C01816=1094.495,429.613,397.808,178.819,24.459,153.656
C01817=1094.490,429.367,397.851,178.817,24.448,153.653
C01818=1094.483,429.120,397.893,178.813,24.437,153.651
C01819=1094.477,428.875,397.935,178.811,24.426,153.649
C01820=1094.470,428.628,397.977,178.808,24.416,153.646
C01821=1094.464,428.382,398.019,178.805,24.405,153.644
C01822=1094.457,428.135,398.061,178.802,24.394,153.642
C01823=1094.451,427.889,398.102,178.799,24.383,153.639
C01824=1094.445,427.643,398.145,178.797,24.373,153.637
C01825=1094.439,427.397,398.186,178.793,24.362,153.635
C01826=1094.433,427.150,398.228,178.791,24.352,153.633
C01827=1094.426,426.904,398.270,178.788,24.342,153.630
C01828=1094.420,426.658,398.312,178.785,24.331,153.628
C01829=1094.413,426.411,398.354,178.782,24.320,153.626
C01830=1094.407,426.165,398.395,178.779,24.310,153.624
C01831=1094.401,425.919,398.437,178.776,24.300,153.622
C01832=1094.395,425.672,398.478,178.774,24.289,153.619
C01833=1094.389,425.443,398.517,178.771,24.280,153.617
C01834=1094.384,425.215,398.556,178.768,24.270,153.615
C01835=1094.378,424.987,398.594,178.766,24.261,153.613
C01836=1094.372,424.758,398.633,178.763,24.251,153.611
C01837=1094.366,424.529,398.671,178.760,24.242,153.609
C01838=1094.360,424.301,398.710,178.757,24.232,153.607
C01839=1094.355,424.073,398.748,178.755,24.223,153.605
C01840=1094.349,423.844,398.787,178.752,24.214,153.603
C01841=1094.344,423.598,398.828,178.749,24.204,153.601
C01842=1094.337,423.351,398.870,178.746,24.194,153.599
C01843=1094.330,423.105,398.911,178.744,24.184,153.597
C01844=1094.324,422.859,398.953,178.741,24.174,153.595
C01845=1094.319,422.612,398.993,178.738,24.164,153.593
C01846=1094.312,422.365,399.035,178.734,24.154,153.591
C01847=1094.306,422.119,399.077,178.732,24.144,153.589
C01848=1094.300,421.873,399.117,178.729,24.134,153.587
C01849=1094.294,421.627,399.158,178.726,24.125,153.585
C01850=1094.287,421.380,399.200,178.723,24.115,153.583
C01851=1094.281,421.134,399.241,178.720,24.105,153.581
C01852=1094.275,420.887,399.282,178.717,24.095,153.579
C01853=1094.269,420.641,399.323,178.714,24.086,153.577
C01854=1094.263,420.393,399.364,178.712,24.076,153.575
C01855=1094.256,420.147,399.405,178.709,24.067,153.573
C01856=1094.250,419.901,399.447,178.706,24.057,153.571
C01857=1094.245,419.654,399.487,178.703,24.048,153.569
C01858=1094.238,419.408,399.528,178.700,24.038,153.567
C01859=1094.232,419.161,399.569,178.697,24.029,153.565
C01860=1094.225,418.914,399.609,178.694,24.019,153.563
C01861=1094.219,418.668,399.651,178.691,24.010,153.561
C01862=1094.214,418.421,399.692,178.689,24.000,153.559
C01863=1094.207,418.175,399.732,178.686,23.991,153.557
C01864=1094.201,417.929,399.773,178.683,23.982,153.555
C01865=1094.195,417.682,399.813,178.680,23.972,153.553
C01866=1094.189,417.436,399.855,178.677,23.963,153.551
C01867=1094.183,417.188,399.896,178.675,23.954,153.549
C01868=1094.176,416.942,399.936,178.672,23.945,153.548
C01869=1094.171,416.695,399.977,178.669,23.936,153.546
C01870=1094.164,416.449,400.018,178.666,23.926,153.544
C01871=1094.158,416.202,400.058,178.663,23.918,153.542
C01872=1094.152,415.956,400.099,178.660,23.908,153.540
C01873=1094.146,415.709,400.139,178.657,23.899,153.538
C01874=1094.140,415.462,400.179,178.654,23.890,153.536
C01875=1094.134,415.216,400.220,178.652,23.882,153.535
C01876=1094.128,414.969,400.260,178.649,23.873,153.533
C01877=1094.122,414.723,400.300,178.646,23.864,153.531
C01878=1094.114,414.476,400.342,178.643,23.855,153.529
C01879=1094.109,414.229,400.382,178.640,23.846,153.527
C01880=1094.102,413.983,400.423,178.636,23.837,153.526
C01881=1094.096,413.735,400.462,178.634,23.828,153.524
C01882=1094.091,413.489,400.503,178.631,23.820,153.522
C01883=1094.084,413.242,400.543,178.628,23.811,153.520
C01884=1094.078,412.996,400.583,178.625,23.802,153.519
C01885=1094.071,412.749,400.623,178.623,23.794,153.517
C01886=1094.066,412.502,400.664,178.620,23.785,153.515
C01887=1094.059,412.256,400.704,178.617,23.776,153.513
C01888=1094.053,412.009,400.744,178.614,23.768,153.512
C01889=1094.048,411.788,400.779,178.611,23.760,153.510
C01890=1094.043,411.567,400.816,178.609,23.753,153.509
C01891=1094.038,411.345,400.852,178.606,23.745,153.507
C01892=1094.032,411.125,400.888,178.604,23.737,153.506
C01893=1094.026,410.904,400.924,178.601,23.730,153.504
C01894=1094.021,410.682,400.959,178.599,23.722,153.503
C01895=1094.015,410.461,400.996,178.595,23.714,153.501
C01896=1094.011,410.240,401.031,178.593,23.706,153.499
C01897=1094.004,409.993,401.071,178.591,23.698,153.498
C01898=1093.998,409.746,401.111,178.588,23.690,153.496
C01899=1093.992,409.500,401.151,178.584,23.681,153.495
C01900=1093.986,409.253,401.192,178.582,23.673,153.493
C01901=1093.980,409.006,401.231,178.579,23.665,153.491
C01902=1093.974,408.759,401.271,178.576,23.656,153.490
C01903=1093.968,408.513,401.310,178.574,23.648,153.488
C01904=1093.962,408.266,401.350,178.570,23.640,153.486
C01905=1093.956,408.019,401.390,178.568,23.632,153.485
C01906=1093.949,407.773,401.430,178.565,23.624,153.483
C01907=1093.943,407.525,401.469,178.561,23.616,153.482
C01908=1093.938,407.279,401.509,178.559,23.607,153.480
C01909=1093.932,407.032,401.549,178.556,23.599,153.478
C01910=1093.926,406.785,401.589,178.554,23.591,153.477
C01911=1093.920,406.538,401.628,178.550,23.583,153.475
C01912=1093.914,406.291,401.668,178.547,23.575,153.474
C01913=1093.908,406.045,401.707,178.545,23.567,153.472
C01914=1093.902,405.798,401.747,178.542,23.559,153.470
C01915=1093.895,405.551,401.786,178.539,23.551,153.469
C01916=1093.889,405.304,401.826,178.536,23.543,153.467
C01917=1093.883,405.058,401.865,178.533,23.536,153.466
C01918=1093.877,404.811,401.904,178.530,23.528,153.464
C01919=1093.871,404.564,401.944,178.528,23.520,153.463
C01920=1093.865,404.317,401.983,178.524,23.512,153.461
C01921=1093.859,404.071,402.023,178.522,23.504,153.460
C01922=1093.853,403.824,402.062,178.519,23.497,153.458
C01923=1093.847,403.577,402.101,178.516,23.489,153.457
C01924=1093.841,403.330,402.140,178.513,23.481,153.455
C01925=1093.835,403.083,402.180,178.510,23.474,153.454
C01926=1093.829,402.836,402.219,178.507,23.466,153.452
C01927=1093.823,402.590,402.258,178.505,23.458,153.451
C01928=1093.817,402.343,402.297,178.501,23.450,153.449
C01929=1093.811,402.096,402.336,178.499,23.443,153.448
C01930=1093.805,401.849,402.375,178.496,23.435,153.446
C01931=1093.799,401.602,402.415,178.493,23.428,153.445
C01932=1093.792,401.355,402.454,178.490,23.421,153.444
C01933=1093.787,401.108,402.492,178.487,23.412,153.442
C01934=1093.781,400.861,402.532,178.485,23.405,153.441
C01935=1093.775,400.614,402.571,178.482,23.398,153.439
C01936=1093.769,400.368,402.609,178.479,23.390,153.438
C01937=1093.763,400.121,402.649,178.476,23.383,153.437
C01938=1093.757,399.874,402.688,178.473,23.376,153.435
C01939=1093.751,399.627,402.726,178.470,23.368,153.434
C01940=1093.745,399.380,402.765,178.468,23.361,153.432
C01941=1093.739,399.133,402.805,178.464,23.353,153.431
C01942=1093.733,398.886,402.843,178.462,23.346,153.430
C01943=1093.727,398.639,402.882,178.459,23.339,153.428
C01944=1093.720,398.393,402.921,178.456,23.332,153.427
C01945=1093.715,398.172,402.956,178.453,23.325,153.426
C01946=1093.710,397.951,402.990,178.451,23.319,153.424
C01947=1093.704,397.730,403.024,178.448,23.312,153.423
C01948=1093.700,397.509,403.059,178.446,23.306,153.422
C01949=1093.694,397.289,403.093,178.443,23.299,153.421
C01950=1093.688,397.068,403.128,178.441,23.293,153.420
C01951=1093.683,396.847,403.163,178.438,23.287,153.418
C01952=1093.678,396.626,403.197,178.435,23.280,153.417
C01953=1093.671,396.379,403.236,178.433,23.274,153.416
C01954=1093.666,396.132,403.274,178.430,23.266,153.415
C01955=1093.659,395.885,403.313,178.427,23.259,153.413
C01956=1093.654,395.638,403.351,178.424,23.252,153.412
C01957=1093.647,395.391,403.390,178.421,23.245,153.411
C01958=1093.642,395.144,403.428,178.418,23.238,153.409
C01959=1093.636,394.898,403.467,178.415,23.231,153.408
C01960=1093.630,394.650,403.506,178.413,23.224,153.407
C01961=1093.624,394.404,403.543,178.410,23.217,153.406
C01962=1093.618,394.157,403.582,178.406,23.210,153.404
C01963=1093.612,393.910,403.621,178.404,23.203,153.403
C01964=1093.606,393.663,403.658,178.401,23.197,153.402
C01965=1093.600,393.416,403.697,178.398,23.190,153.401
C01966=1093.594,393.169,403.735,178.395,23.183,153.399
C01967=1093.588,392.922,403.774,178.392,23.176,153.398
C01968=1093.582,392.675,403.811,178.389,23.169,153.397
C01969=1093.576,392.428,403.849,178.387,23.163,153.396
C01970=1093.570,392.181,403.889,178.384,23.156,153.394
C01971=1093.564,391.934,403.926,178.380,23.149,153.393
C01972=1093.558,391.688,403.964,178.378,23.142,153.392
C01973=1093.552,391.440,404.002,178.375,23.136,153.391
C01974=1093.546,391.193,404.040,178.372,23.130,153.390
C01975=1093.540,390.947,404.078,178.369,23.123,153.388
C01976=1093.534,390.699,404.116,178.366,23.116,153.387
C01977=1093.528,390.452,404.154,178.363,23.110,153.386
C01978=1093.522,390.206,404.193,178.360,23.103,153.385
C01979=1093.516,389.959,404.231,178.357,23.096,153.384
C01980=1093.510,389.712,404.268,178.355,23.090,153.383
C01981=1093.504,389.465,404.306,178.351,23.083,153.381
C01982=1093.498,389.218,404.344,178.348,23.076,153.380
C01983=1093.491,388.971,404.382,178.345,23.070,153.379
C01984=1093.486,388.724,404.419,178.343,23.064,153.378
C01985=1093.480,388.477,404.457,178.340,23.057,153.377
C01986=1093.474,388.230,404.495,178.337,23.051,153.376
C01987=1093.468,387.983,404.532,178.333,23.044,153.375
C01988=1093.462,387.736,404.571,178.331,23.038,153.373
C01989=1093.456,387.489,404.608,178.328,23.031,153.372
C01990=1093.450,387.242,404.646,178.325,23.025,153.371
C01991=1093.444,386.995,404.683,178.322,23.019,153.370
C01992=1093.438,386.748,404.721,178.319,23.013,153.369
C01993=1093.432,386.502,404.759,178.316,23.006,153.368
C01994=1093.426,386.254,404.797,178.314,23.000,153.367
C01995=1093.420,386.007,404.834,178.310,22.993,153.366
C01996=1093.414,385.760,404.872,178.307,22.987,153.365
C01997=1093.408,385.513,404.909,178.304,22.981,153.363
C01998=1093.402,385.267,404.947,178.301,22.975,153.362
C01999=1093.397,385.019,404.984,178.298,22.969,153.361
C02000=1093.391,384.772,405.022,178.296,22.962,153.360
C02001=1093.386,384.558,405.054,178.294,22.957,153.359
C02002=1093.381,384.343,405.087,178.290,22.951,153.358
C02003=1093.376,384.129,405.120,178.288,22.946,153.357
C02004=1093.371,383.915,405.152,178.285,22.940,153.356
C02005=1093.365,383.700,405.184,178.283,22.935,153.356
C02006=1093.361,383.486,405.217,178.281,22.930,153.355
C02007=1093.355,383.272,405.249,178.278,22.924,153.354
C02008=1093.351,383.057,405.281,178.276,22.919,153.353
C02009=1093.345,382.811,405.319,178.273,22.913,153.352
C02010=1093.339,382.563,405.356,178.270,22.907,153.351
C02011=1093.332,382.316,405.393,178.267,22.901,153.350
C02012=1093.326,382.069,405.431,178.264,22.895,153.349
C02013=1093.321,381.821,405.468,178.261,22.889,153.348
C02014=1093.314,381.575,405.505,178.258,22.883,153.347
C02015=1093.308,381.328,405.542,178.255,22.877,153.346
C02016=1093.303,381.080,405.579,178.252,22.871,153.345
C02017=1093.296,380.834,405.616,178.249,22.866,153.344
C02018=1093.291,380.587,405.653,178.245,22.859,153.343
C02019=1093.285,380.339,405.690,178.242,22.853,153.342
C02020=1093.278,380.093,405.727,178.239,22.847,153.341
C02021=1093.273,379.845,405.764,178.237,22.841,153.340
C02022=1093.267,379.598,405.801,178.234,22.836,153.339
C02023=1093.261,379.351,405.838,178.231,22.830,153.338
C02024=1093.255,379.104,405.875,178.228,22.824,153.337
C02025=1093.249,378.857,405.913,178.226,22.818,153.336
C02026=1093.243,378.610,405.949,178.222,22.813,153.335
C02027=1093.237,378.362,405.986,178.219,22.807,153.334
C02028=1093.231,378.115,406.023,178.217,22.801,153.333
C02029=1093.225,377.868,406.060,178.213,22.796,153.332
C02030=1093.220,377.621,406.097,178.210,22.790,153.331
C02031=1093.213,377.374,406.133,178.208,22.784,153.330
C02032=1093.208,377.127,406.170,178.204,22.778,153.329
C02033=1093.202,376.880,406.206,178.202,22.772,153.328
C02034=1093.197,376.633,406.243,178.198,22.767,153.327
C02035=1093.191,376.385,406.280,178.196,22.761,153.326
C02036=1093.185,376.138,406.317,178.192,22.755,153.325
C02037=1093.179,375.891,406.354,178.189,22.749,153.324
C02038=1093.173,375.644,406.390,178.186,22.744,153.323
C02039=1093.167,375.396,406.427,178.183,22.738,153.323
C02040=1093.161,375.150,406.463,178.180,22.732,153.322
C02041=1093.156,374.903,406.500,178.177,22.727,153.321
C02042=1093.149,374.656,406.537,178.175,22.722,153.320
C02043=1093.144,374.408,406.574,178.172,22.716,153.319
C02044=1093.138,374.160,406.610,178.169,22.710,153.318
C02045=1093.132,373.913,406.647,178.166,22.705,153.317
C02046=1093.126,373.666,406.683,178.163,22.699,153.316
C02047=1093.120,373.420,406.719,178.160,22.694,153.315
C02048=1093.115,373.172,406.756,178.157,22.688,153.315
C02049=1093.108,372.925,406.792,178.154,22.683,153.314
C02050=1093.102,372.678,406.828,178.150,22.677,153.313
C02051=1093.096,372.431,406.865,178.147,22.672,153.312
C02052=1093.091,372.183,406.901,178.145,22.667,153.311
C02053=1093.084,371.936,406.938,178.142,22.661,153.310
C02054=1093.078,371.689,406.974,178.139,22.656,153.309
C02055=1093.073,371.441,407.010,178.136,22.650,153.309
C02056=1093.067,371.194,407.047,178.133,22.645,153.308
C02057=1093.057,370.793,407.105,178.128,22.636,153.306
C02058=1093.048,370.391,407.164,178.123,22.627,153.305
C02059=1093.038,369.990,407.223,178.119,22.619,153.304
C02060=1093.029,369.590,407.281,178.114,22.610,153.302
C02061=1093.023,369.342,407.317,178.111,22.605,153.301
C02062=1093.017,369.094,407.353,178.107,22.600,153.301
C02063=1093.011,368.847,407.390,178.104,22.594,153.300
C02064=1093.005,368.600,407.425,178.101,22.589,153.299
C02065=1092.999,368.353,407.462,178.099,22.584,153.298
C02066=1092.993,368.105,407.497,178.096,22.579,153.297
C02067=1092.988,367.858,407.533,178.092,22.574,153.297
C02068=1092.982,367.611,407.570,178.089,22.568,153.296
C02069=1092.976,367.363,407.606,178.086,22.563,153.295
C02070=1092.971,367.116,407.641,178.084,22.558,153.294
C02071=1092.964,366.869,407.677,178.081,22.553,153.293
C02072=1092.958,366.622,407.713,178.077,22.548,153.293
C02073=1092.954,366.374,407.749,178.074,22.542,153.292
C02074=1092.948,366.127,407.785,178.071,22.537,153.291
C02075=1092.941,365.880,407.821,178.069,22.532,153.290
C02076=1092.936,365.633,407.857,178.066,22.527,153.289
C02077=1092.930,365.385,407.892,178.062,22.522,153.289
C02078=1092.924,365.137,407.928,178.059,22.517,153.288
C02079=1092.918,364.890,407.963,178.056,22.512,153.287
C02080=1092.912,364.643,408.000,178.054,22.507,153.287
C02081=1092.906,364.396,408.036,178.050,22.502,153.286
C02082=1092.900,364.149,408.071,178.047,22.497,153.285
C02083=1092.894,363.901,408.107,178.044,22.491,153.284
C02084=1092.889,363.654,408.142,178.042,22.487,153.284
C02085=1092.883,363.406,408.178,178.038,22.482,153.283
C02086=1092.876,363.159,408.213,178.035,22.477,153.282
C02087=1092.871,362.912,408.248,178.032,22.471,153.281
C02088=1092.865,362.664,408.284,178.029,22.467,153.281
C02089=1092.859,362.417,408.319,178.026,22.462,153.280
C02090=1092.853,362.170,408.355,178.023,22.457,153.279
C02091=1092.847,361.922,408.391,178.020,22.452,153.279
C02092=1092.842,361.675,408.426,178.017,22.447,153.278
C02093=1092.836,361.427,408.462,178.014,22.442,153.277
C02094=1092.831,361.180,408.497,178.011,22.437,153.276
C02095=1092.824,360.932,408.532,178.008,22.433,153.276
C02096=1092.818,360.685,408.567,178.005,22.428,153.275
C02097=1092.812,360.438,408.603,178.002,22.423,153.274
C02098=1092.807,360.191,408.638,177.999,22.418,153.274
C02099=1092.801,359.943,408.674,177.996,22.414,153.273
C02100=1092.795,359.695,408.708,177.993,22.408,153.272
C02101=1092.789,359.448,408.744,177.990,22.403,153.271
C02102=1092.783,359.200,408.779,177.987,22.399,153.271
C02103=1092.778,358.953,408.815,177.984,22.394,153.270
C02104=1092.771,358.705,408.849,177.980,22.389,153.270
C02105=1092.766,358.458,408.885,177.978,22.385,153.269
C02106=1092.760,358.211,408.920,177.975,22.380,153.268
C02107=1092.754,357.963,408.954,177.971,22.375,153.267
C02108=1092.748,357.716,408.990,177.969,22.371,153.267
C02109=1092.739,357.330,409.045,177.963,22.363,153.266
C02110=1092.730,356.944,409.099,177.959,22.356,153.265
C02111=1092.721,356.558,409.154,177.955,22.349,153.264
C02112=1092.712,356.172,409.209,177.950,22.342,153.263
C02113=1092.706,355.925,409.243,177.947,22.337,153.262
C02114=1092.700,355.678,409.278,177.943,22.332,153.261
C02115=1092.695,355.429,409.313,177.941,22.328,153.261
C02116=1092.688,355.183,409.348,177.937,22.323,153.260
C02117=1092.683,354.935,409.383,177.934,22.318,153.260
C02118=1092.677,354.688,409.418,177.932,22.314,153.259
C02119=1092.671,354.440,409.453,177.928,22.309,153.258
C02120=1092.666,354.192,409.488,177.925,22.304,153.258
C02121=1092.659,353.945,409.522,177.922,22.300,153.257
C02122=1092.654,353.697,409.557,177.919,22.295,153.256
C02123=1092.648,353.449,409.592,177.916,22.291,153.256
C02124=1092.642,353.203,409.627,177.913,22.286,153.255
C02125=1092.637,352.955,409.661,177.910,22.282,153.255
C02126=1092.631,352.707,409.696,177.907,22.277,153.254
C02127=1092.625,352.460,409.731,177.904,22.273,153.253
C02128=1092.619,352.212,409.766,177.901,22.269,153.253
C02129=1092.613,351.965,409.800,177.898,22.264,153.252
C02130=1092.608,351.717,409.834,177.894,22.259,153.252
C02131=1092.601,351.470,409.870,177.892,22.255,153.251
C02132=1092.595,351.222,409.904,177.889,22.250,153.250
C02133=1092.586,350.816,409.960,177.884,22.243,153.249
C02134=1092.576,350.409,410.017,177.879,22.236,153.249
C02135=1092.566,350.002,410.074,177.874,22.229,153.248
C02136=1092.557,349.596,410.130,177.869,22.221,153.247
C02137=1092.552,349.348,410.165,177.865,22.217,153.246
C02138=1092.546,349.101,410.199,177.863,22.213,153.245
C02139=1092.540,348.853,410.233,177.859,22.208,153.245
C02140=1092.534,348.605,410.268,177.856,22.204,153.244
C02141=1092.529,348.358,410.302,177.853,22.199,153.244
C02142=1092.523,348.111,410.336,177.851,22.195,153.243
C02143=1092.518,347.863,410.371,177.847,22.191,153.243
C02144=1092.511,347.615,410.405,177.844,22.187,153.242
C02145=1092.505,347.368,410.439,177.841,22.182,153.242
C02146=1092.500,347.120,410.474,177.838,22.178,153.241
C02147=1092.494,346.873,410.508,177.835,22.174,153.241
C02148=1092.488,346.625,410.542,177.832,22.169,153.240
C02149=1092.482,346.377,410.576,177.829,22.165,153.239
C02150=1092.477,346.129,410.610,177.825,22.161,153.239
C02151=1092.471,345.882,410.644,177.823,22.157,153.238
C02152=1092.465,345.635,410.678,177.819,22.152,153.238
C02153=1092.459,345.387,410.713,177.817,22.148,153.237
C02154=1092.453,345.139,410.746,177.813,22.144,153.237
C02155=1092.448,344.891,410.781,177.811,22.140,153.236
C02156=1092.442,344.644,410.815,177.807,22.135,153.236
C02157=1092.436,344.408,410.847,177.805,22.132,153.235
C02158=1092.431,344.172,410.880,177.802,22.128,153.235
C02159=1092.426,343.935,410.912,177.798,22.124,153.234
C02160=1092.420,343.700,410.944,177.796,22.119,153.234
C02161=1092.414,343.464,410.977,177.793,22.116,153.233
C02162=1092.408,343.229,411.009,177.790,22.112,153.233
C02163=1092.403,342.992,411.041,177.787,22.108,153.232
C02164=1092.398,342.756,411.073,177.784,22.104,153.232
C02165=1092.392,342.509,411.107,177.781,22.100,153.231
C02166=1092.386,342.260,411.141,177.778,22.096,153.231
C02167=1092.380,342.013,411.175,177.775,22.092,153.230
C02168=1092.375,341.765,411.208,177.772,22.088,153.230
C02169=1092.369,341.518,411.242,177.769,22.084,153.229
C02170=1092.363,341.270,411.276,177.766,22.079,153.229
C02171=1092.357,341.023,411.310,177.763,22.075,153.228
C02172=1092.352,340.775,411.343,177.759,22.071,153.228
C02173=1092.346,340.527,411.377,177.757,22.067,153.227
C02174=1092.340,340.280,411.411,177.753,22.063,153.227
C02175=1092.334,340.032,411.445,177.751,22.059,153.226
C02176=1092.328,339.784,411.478,177.747,22.055,153.226
C02177=1092.322,339.536,411.512,177.744,22.051,153.225
C02178=1092.317,339.288,411.546,177.742,22.047,153.225
C02179=1092.311,339.041,411.579,177.738,22.043,153.225
C02180=1092.305,338.793,411.613,177.735,22.039,153.224
C02181=1092.300,338.545,411.646,177.732,22.035,153.224
C02182=1092.294,338.298,411.679,177.729,22.031,153.223
C02183=1092.288,338.051,411.713,177.726,22.027,153.223
C02184=1092.282,337.803,411.747,177.723,22.023,153.222
C02185=1092.277,337.555,411.780,177.720,22.019,153.222
C02186=1092.271,337.307,411.813,177.717,22.015,153.221
C02187=1092.265,337.060,411.847,177.714,22.011,153.221
C02188=1092.259,336.812,411.880,177.710,22.007,153.220
C02189=1092.253,336.564,411.913,177.708,22.003,153.220
C02190=1092.248,336.316,411.947,177.704,21.999,153.220
C02191=1092.242,336.068,411.980,177.701,21.995,153.219
C02192=1092.236,335.821,412.014,177.698,21.992,153.219
C02193=1092.230,335.573,412.047,177.695,21.988,153.218
C02194=1092.225,335.325,412.080,177.692,21.984,153.218
C02195=1092.219,335.078,412.114,177.689,21.980,153.217
C02196=1092.213,334.830,412.146,177.686,21.976,153.217
C02197=1092.207,334.582,412.180,177.683,21.972,153.216
C02198=1092.202,334.334,412.213,177.680,21.969,153.216
C02199=1092.195,334.087,412.246,177.677,21.965,153.216
C02200=1092.190,333.839,412.279,177.674,21.961,153.215
C02201=1092.184,333.591,412.312,177.671,21.957,153.215
C02202=1092.179,333.343,412.346,177.668,21.954,153.214
C02203=1092.172,333.095,412.378,177.664,21.949,153.214
C02204=1092.167,332.848,412.411,177.661,21.946,153.214
C02205=1092.162,332.600,412.445,177.659,21.942,153.213
C02206=1092.156,332.353,412.478,177.655,21.938,153.213
C02207=1092.150,332.105,412.511,177.652,21.934,153.212
C02208=1092.144,331.857,412.544,177.650,21.930,153.212
C02209=1092.138,331.609,412.577,177.646,21.927,153.212
C02210=1092.132,331.362,412.610,177.643,21.923,153.211
C02211=1092.126,331.114,412.643,177.640,21.920,153.211
C02212=1092.120,330.866,412.676,177.637,21.915,153.210
C02213=1092.111,330.477,412.727,177.632,21.910,153.210
C02214=1092.102,330.087,412.778,177.628,21.905,153.209
C02215=1092.093,329.698,412.830,177.623,21.898,153.209
C02216=1092.083,329.308,412.881,177.618,21.893,153.208
C02217=1092.078,329.061,412.915,177.615,21.889,153.208
C02218=1092.072,328.813,412.947,177.611,21.885,153.207
C02219=1092.066,328.565,412.979,177.608,21.882,153.207
C02220=1092.061,328.318,413.012,177.605,21.879,153.207
C02221=1092.054,328.070,413.045,177.602,21.874,153.206
C02222=1092.049,327.821,413.078,177.599,21.871,153.206
C02223=1092.043,327.574,413.111,177.596,21.868,153.205
C02224=1092.036,327.326,413.143,177.593,21.864,153.205
C02225=1092.031,327.078,413.176,177.590,21.860,153.205
C02226=1092.026,326.831,413.208,177.587,21.857,153.204
C02227=1092.020,326.583,413.240,177.584,21.853,153.204
C02228=1092.014,326.335,413.274,177.580,21.849,153.204
C02229=1092.008,326.086,413.306,177.577,21.846,153.203
C02230=1092.002,325.839,413.338,177.575,21.842,153.203
C02231=1091.996,325.592,413.371,177.571,21.838,153.203
C02232=1091.991,325.343,413.403,177.568,21.835,153.202
C02233=1091.984,325.096,413.436,177.565,21.832,153.202
C02234=1091.978,324.848,413.468,177.563,21.828,153.201
C02235=1091.974,324.600,413.500,177.559,21.824,153.201
C02236=1091.968,324.352,413.533,177.556,21.821,153.201
C02237=1091.962,324.104,413.565,177.553,21.817,153.200
C02238=1091.956,323.857,413.598,177.550,21.814,153.200
C02239=1091.951,323.609,413.630,177.547,21.810,153.200
C02240=1091.945,323.360,413.662,177.544,21.807,153.199
C02241=1091.938,323.113,413.695,177.541,21.803,153.199
C02242=1091.933,322.865,413.727,177.538,21.800,153.199
C02243=1091.927,322.617,413.760,177.534,21.796,153.198
C02244=1091.921,322.369,413.792,177.532,21.792,153.198
C02245=1091.916,322.122,413.824,177.529,21.789,153.198
C02246=1091.910,321.873,413.856,177.526,21.786,153.197
C02247=1091.904,321.626,413.889,177.522,21.782,153.197
C02248=1091.899,321.378,413.921,177.519,21.779,153.197
C02249=1091.893,321.130,413.953,177.517,21.775,153.196
C02250=1091.888,320.882,413.984,177.514,21.772,153.196
C02251=1091.881,320.635,414.017,177.510,21.768,153.196
C02252=1091.876,320.386,414.050,177.507,21.764,153.195
C02253=1091.871,320.139,414.081,177.504,21.761,153.195
C02254=1091.865,319.890,414.113,177.502,21.758,153.195
C02255=1091.859,319.643,414.145,177.498,21.754,153.194
C02256=1091.853,319.395,414.177,177.495,21.751,153.194
C02257=1091.848,319.148,414.210,177.492,21.747,153.194
C02258=1091.842,318.900,414.242,177.489,21.744,153.193
C02259=1091.837,318.651,414.274,177.486,21.741,153.193
C02260=1091.831,318.404,414.306,177.483,21.737,153.193
C02261=1091.825,318.155,414.338,177.480,21.733,153.192
C02262=1091.820,317.908,414.370,177.477,21.730,153.192
C02263=1091.814,317.660,414.402,177.474,21.727,153.192
C02264=1091.808,317.412,414.433,177.470,21.723,153.191
C02265=1091.799,317.016,414.485,177.466,21.718,153.191
C02266=1091.791,316.620,414.535,177.461,21.712,153.190
C02267=1091.782,316.224,414.587,177.456,21.706,153.190
C02268=1091.773,315.827,414.637,177.452,21.702,153.189
C02269=1091.767,315.579,414.669,177.448,21.698,153.189
C02270=1091.761,315.332,414.700,177.445,21.694,153.189
C02271=1091.755,315.083,414.732,177.442,21.691,153.189
C02272=1091.750,314.836,414.764,177.439,21.688,153.188
C02273=1091.744,314.587,414.795,177.436,21.685,153.188
C02274=1091.739,314.339,414.827,177.433,21.682,153.188
C02275=1091.732,314.092,414.858,177.430,21.678,153.187
C02276=1091.727,313.844,414.890,177.427,21.675,153.187
C02277=1091.721,313.596,414.922,177.424,21.672,153.187
C02278=1091.715,313.347,414.953,177.421,21.668,153.187
C02279=1091.709,313.100,414.984,177.418,21.665,153.186
C02280=1091.703,312.852,415.016,177.415,21.662,153.186
C02281=1091.698,312.604,415.048,177.411,21.659,153.186
C02282=1091.691,312.356,415.079,177.408,21.655,153.186
C02283=1091.686,312.108,415.110,177.405,21.652,153.185
C02284=1091.680,311.861,415.142,177.402,21.649,153.185
C02285=1091.674,311.612,415.173,177.399,21.646,153.185
C02286=1091.669,311.364,415.205,177.396,21.643,153.185
C02287=1091.663,311.116,415.237,177.393,21.639,153.184
C02288=1091.657,310.868,415.267,177.390,21.636,153.184
C02289=1091.651,310.620,415.299,177.387,21.633,153.184
C02290=1091.645,310.373,415.331,177.384,21.630,153.183
C02291=1091.640,310.125,415.361,177.381,21.627,153.183
C02292=1091.634,309.877,415.393,177.378,21.623,153.183
C02293=1091.628,309.629,415.423,177.375,21.621,153.183
C02294=1091.622,309.381,415.455,177.371,21.617,153.183
C02295=1091.617,309.133,415.486,177.368,21.614,153.182
C02296=1091.611,308.885,415.517,177.365,21.611,153.182
C02297=1091.605,308.636,415.549,177.362,21.608,153.182
C02298=1091.599,308.389,415.580,177.359,21.604,153.182
C02299=1091.594,308.141,415.611,177.356,21.602,153.181
C02300=1091.588,307.893,415.643,177.353,21.598,153.181
C02301=1091.582,307.645,415.673,177.350,21.595,153.181
C02302=1091.577,307.398,415.705,177.347,21.591,153.181
C02303=1091.570,307.149,415.735,177.344,21.589,153.180
C02304=1091.565,306.902,415.767,177.341,21.585,153.180
C02305=1091.559,306.654,415.797,177.338,21.582,153.180
C02306=1091.553,306.405,415.829,177.335,21.579,153.180
C02307=1091.547,306.158,415.860,177.332,21.576,153.179
C02308=1091.542,305.910,415.891,177.329,21.573,153.179
C02309=1091.537,305.661,415.922,177.326,21.570,153.179
C02310=1091.530,305.414,415.953,177.322,21.567,153.179
C02311=1091.525,305.165,415.984,177.319,21.563,153.178
C02312=1091.519,304.918,416.014,177.316,21.560,153.178
C02313=1091.514,304.669,416.045,177.313,21.557,153.178
C02314=1091.508,304.422,416.077,177.310,21.554,153.178
C02315=1091.502,304.173,416.108,177.307,21.551,153.177
C02316=1091.497,303.926,416.138,177.304,21.548,153.177
C02317=1091.488,303.532,416.187,177.299,21.543,153.177
C02318=1091.479,303.138,416.237,177.295,21.538,153.176
C02319=1091.470,302.746,416.285,177.289,21.533,153.176
C02320=1091.461,302.352,416.333,177.285,21.528,153.176
C02321=1091.455,302.103,416.364,177.282,21.525,153.175
C02322=1091.449,301.856,416.396,177.279,21.522,153.175
C02323=1091.444,301.608,416.426,177.275,21.519,153.175
C02324=1091.439,301.360,416.457,177.272,21.515,153.175
C02325=1091.433,301.112,416.487,177.269,21.513,153.175
C02326=1091.427,300.864,416.518,177.266,21.509,153.174
C02327=1091.422,300.616,416.549,177.263,21.506,153.174
C02328=1091.416,300.368,416.579,177.260,21.503,153.174
C02329=1091.410,300.119,416.610,177.257,21.500,153.174
C02330=1091.405,299.871,416.641,177.254,21.497,153.173
C02331=1091.399,299.624,416.671,177.251,21.494,153.173
C02332=1091.394,299.376,416.702,177.248,21.491,153.173
C02333=1091.388,299.128,416.732,177.245,21.488,153.173
C02334=1091.383,298.880,416.763,177.242,21.485,153.173
C02335=1091.377,298.631,416.793,177.239,21.482,153.172
C02336=1091.371,298.383,416.823,177.236,21.479,153.172
C02337=1091.366,298.135,416.854,177.233,21.476,153.172
C02338=1091.361,297.887,416.885,177.231,21.473,153.172
C02339=1091.355,297.640,416.915,177.227,21.469,153.171
C02340=1091.349,297.392,416.945,177.224,21.467,153.171
C02341=1091.342,297.143,416.976,177.221,21.464,153.171
C02342=1091.337,296.895,417.006,177.218,21.461,153.171
C02343=1091.332,296.647,417.037,177.214,21.458,153.171
C02344=1091.326,296.399,417.067,177.211,21.455,153.171
C02345=1091.320,296.151,417.097,177.209,21.452,153.170
C02346=1091.315,295.903,417.127,177.206,21.449,153.170
C02347=1091.309,295.655,417.157,177.202,21.446,153.170
C02348=1091.303,295.407,417.188,177.199,21.443,153.170
C02349=1091.297,295.159,417.218,177.196,21.440,153.170
C02350=1091.292,294.911,417.248,177.193,21.437,153.169
C02351=1091.286,294.663,417.278,177.190,21.434,153.169
C02352=1091.280,294.415,417.308,177.187,21.431,153.169
C02353=1091.275,294.167,417.338,177.184,21.429,153.169
C02354=1091.269,293.919,417.368,177.181,21.426,153.169
C02355=1091.263,293.670,417.398,177.178,21.423,153.169
C02356=1091.257,293.422,417.428,177.175,21.420,153.168
C02357=1091.252,293.174,417.459,177.172,21.417,153.168
C02358=1091.247,292.926,417.489,177.169,21.414,153.168
C02359=1091.241,292.678,417.519,177.166,21.411,153.168
C02360=1091.236,292.430,417.549,177.163,21.408,153.168
C02361=1091.230,292.182,417.579,177.160,21.406,153.167
C02362=1091.224,291.934,417.608,177.157,21.403,153.167
C02363=1091.218,291.686,417.639,177.154,21.400,153.167
C02364=1091.212,291.437,417.668,177.151,21.397,153.167
C02365=1091.206,291.190,417.699,177.148,21.394,153.167
C02366=1091.201,290.941,417.728,177.145,21.391,153.167
C02367=1091.195,290.693,417.759,177.142,21.388,153.166
C02368=1091.190,290.445,417.788,177.139,21.385,153.166
C02369=1091.181,290.065,417.834,177.134,21.381,153.166
C02370=1091.172,289.686,417.879,177.129,21.377,153.166
C02371=1091.164,289.306,417.925,177.125,21.372,153.165
C02372=1091.155,288.927,417.971,177.120,21.368,153.165
C02373=1091.149,288.679,418.000,177.117,21.365,153.165
C02374=1091.144,288.430,418.030,177.114,21.362,153.165
C02375=1091.137,288.182,418.059,177.111,21.359,153.165
C02376=1091.132,287.934,418.089,177.108,21.356,153.165
C02377=1091.126,287.686,418.119,177.105,21.354,153.165
C02378=1091.121,287.437,418.149,177.102,21.351,153.164
C02379=1091.114,287.189,418.178,177.099,21.348,153.164
C02380=1091.108,286.942,418.208,177.096,21.345,153.164
C02381=1091.103,286.693,418.238,177.093,21.342,153.164
C02382=1091.098,286.445,418.267,177.090,21.340,153.164
C02383=1091.092,286.197,418.296,177.087,21.337,153.163
C02384=1091.086,285.949,418.326,177.083,21.334,153.163
C02385=1091.080,285.701,418.356,177.080,21.331,153.163
C02386=1091.075,285.453,418.386,177.077,21.328,153.163
C02387=1091.069,285.204,418.415,177.074,21.326,153.163
C02388=1091.063,284.956,418.444,177.071,21.323,153.163
C02389=1091.058,284.708,418.474,177.069,21.320,153.163
C02390=1091.052,284.460,418.503,177.066,21.318,153.163
C02391=1091.047,284.212,418.532,177.063,21.315,153.162
C02392=1091.041,283.963,418.562,177.060,21.312,153.162
C02393=1091.035,283.715,418.591,177.057,21.309,153.162
C02394=1091.030,283.467,418.620,177.054,21.306,153.162
C02395=1091.024,283.219,418.650,177.051,21.303,153.162
C02396=1091.018,282.971,418.679,177.048,21.301,153.162
C02397=1091.013,282.722,418.709,177.044,21.298,153.161
C02398=1091.007,282.474,418.738,177.041,21.295,153.161
C02399=1091.001,282.226,418.767,177.038,21.292,153.161
C02400=1090.996,281.978,418.796,177.035,21.289,153.161
C02401=1090.990,281.730,418.826,177.032,21.287,153.161
C02402=1090.984,281.481,418.855,177.029,21.284,153.161
C02403=1090.979,281.234,418.884,177.027,21.282,153.161
C02404=1090.973,280.986,418.913,177.024,21.279,153.160
C02405=1090.968,280.736,418.942,177.021,21.276,153.160
C02406=1090.962,280.488,418.971,177.018,21.273,153.160
C02407=1090.957,280.241,419.001,177.015,21.271,153.160
C02408=1090.950,279.992,419.030,177.011,21.268,153.160
C02409=1090.945,279.744,419.059,177.008,21.265,153.160
C02410=1090.939,279.495,419.088,177.005,21.262,153.160
C02411=1090.934,279.248,419.117,177.002,21.259,153.159
C02412=1090.928,278.999,419.146,176.999,21.257,153.159
C02413=1090.922,278.751,419.176,176.997,21.255,153.159
C02414=1090.917,278.503,419.204,176.994,21.252,153.159
C02415=1090.911,278.255,419.233,176.991,21.249,153.159
C02416=1090.905,278.006,419.262,176.988,21.246,153.159
C02417=1090.899,277.758,419.291,176.985,21.244,153.159
C02418=1090.894,277.510,419.320,176.981,21.241,153.159
C02419=1090.888,277.262,419.349,176.978,21.238,153.159
C02420=1090.883,277.013,419.379,176.975,21.235,153.158
C02421=1090.874,276.643,419.421,176.970,21.231,153.158
C02422=1090.866,276.273,419.464,176.967,21.228,153.158
C02423=1090.857,275.903,419.507,176.962,21.224,153.158
C02424=1090.848,275.533,419.550,176.957,21.220,153.158
C02425=1090.843,275.285,419.579,176.954,21.217,153.158
C02426=1090.838,275.036,419.607,176.951,21.214,153.157
C02427=1090.831,274.788,419.636,176.949,21.212,153.157
C02428=1090.827,274.540,419.665,176.946,21.209,153.157
C02429=1090.820,274.292,419.694,176.943,21.206,153.157
C02430=1090.815,274.044,419.722,176.940,21.204,153.157
C02431=1090.809,273.795,419.751,176.937,21.201,153.157
C02432=1090.804,273.546,419.780,176.933,21.199,153.157
C02433=1090.798,273.298,419.808,176.930,21.196,153.157
C02434=1090.792,273.050,419.837,176.928,21.194,153.157
C02435=1090.787,272.802,419.865,176.925,21.191,153.156
C02436=1090.781,272.554,419.894,176.922,21.188,153.156
C02437=1090.775,272.305,419.923,176.919,21.185,153.156
C02438=1090.770,272.057,419.951,176.916,21.183,153.156
C02439=1090.764,271.809,419.980,176.912,21.180,153.156
C02440=1090.758,271.561,420.008,176.909,21.177,153.156
C02441=1090.752,271.312,420.036,176.907,21.175,153.156
C02442=1090.747,271.064,420.066,176.904,21.172,153.156
C02443=1090.741,270.816,420.094,176.901,21.170,153.156
C02444=1090.736,270.567,420.122,176.898,21.167,153.155
C02445=1090.730,270.319,420.151,176.894,21.165,153.155
C02446=1090.724,270.071,420.179,176.891,21.162,153.155
C02447=1090.719,269.823,420.207,176.889,21.160,153.155
C02448=1090.713,269.574,420.235,176.886,21.157,153.155
C02449=1090.708,269.325,420.264,176.883,21.154,153.155
C02450=1090.702,269.077,420.293,176.880,21.152,153.155
C02451=1090.696,268.829,420.321,176.876,21.149,153.155
C02452=1090.691,268.580,420.349,176.873,21.146,153.155
C02453=1090.685,268.332,420.377,176.871,21.144,153.155
C02454=1090.679,268.084,420.405,176.868,21.141,153.154
C02455=1090.673,267.835,420.434,176.865,21.139,153.154
C02456=1090.668,267.587,420.462,176.862,21.136,153.154
C02457=1090.662,267.339,420.491,176.859,21.134,153.154
C02458=1090.656,267.091,420.519,176.856,21.131,153.154
C02459=1090.651,266.843,420.547,176.853,21.129,153.154
C02460=1090.645,266.594,420.575,176.850,21.126,153.154
C02461=1090.640,266.346,420.603,176.847,21.123,153.154
C02462=1090.634,266.097,420.631,176.844,21.121,153.154
C02463=1090.628,265.849,420.659,176.841,21.118,153.154
C02464=1090.623,265.600,420.688,176.838,21.116,153.153
C02465=1090.617,265.352,420.716,176.835,21.113,153.153
C02466=1090.611,265.103,420.744,176.832,21.111,153.153
C02467=1090.606,264.855,420.772,176.829,21.108,153.153
C02468=1090.601,264.607,420.800,176.826,21.105,153.153
C02469=1090.595,264.359,420.828,176.824,21.103,153.153
C02470=1090.589,264.111,420.855,176.820,21.101,153.153
C02471=1090.583,263.862,420.884,176.817,21.098,153.153
C02472=1090.577,263.614,420.912,176.814,21.095,153.153
C02473=1090.569,263.246,420.953,176.810,21.092,153.153
C02474=1090.560,262.879,420.994,176.805,21.088,153.153
C02475=1090.551,262.512,421.034,176.801,21.084,153.152
C02476=1090.543,262.145,421.076,176.797,21.081,153.152
C02477=1090.537,261.896,421.104,176.794,21.078,153.152
C02478=1090.531,261.648,421.132,176.790,21.076,153.152
C02479=1090.526,261.399,421.159,176.787,21.073,153.152
C02480=1090.520,261.151,421.187,176.785,21.071,153.152
C02481=1090.514,260.903,421.215,176.782,21.069,153.152
C02482=1090.508,260.654,421.243,176.779,21.066,153.152
C02483=1090.502,260.405,421.270,176.776,21.063,153.152
C02484=1090.497,260.157,421.298,176.773,21.061,153.152
C02485=1090.491,259.909,421.326,176.770,21.059,153.152
C02486=1090.485,259.660,421.353,176.767,21.056,153.152
C02487=1090.479,259.412,421.381,176.764,21.054,153.152
C02488=1090.474,259.163,421.409,176.761,21.052,153.152
C02489=1090.468,258.915,421.436,176.758,21.049,153.152
C02490=1090.462,258.666,421.464,176.755,21.046,153.151
C02491=1090.457,258.418,421.492,176.752,21.044,153.151
C02492=1090.451,258.170,421.519,176.749,21.041,153.151
C02493=1090.445,257.921,421.547,176.746,21.039,153.151
C02494=1090.440,257.673,421.574,176.743,21.037,153.151
C02495=1090.434,257.425,421.602,176.740,21.034,153.151
C02496=1090.429,257.175,421.629,176.737,21.032,153.151
C02497=1090.422,256.928,421.657,176.735,21.029,153.151
C02498=1090.417,256.679,421.684,176.731,21.027,153.151
C02499=1090.411,256.431,421.711,176.728,21.024,153.151
C02500=1090.406,256.182,421.739,176.725,21.021,153.151
C02501=1090.400,255.934,421.767,176.723,21.019,153.151
C02502=1090.395,255.685,421.794,176.720,21.017,153.151
C02503=1090.389,255.437,421.822,176.716,21.014,153.150
C02504=1090.383,255.188,421.849,176.713,21.012,153.150
C02505=1090.378,254.940,421.877,176.711,21.010,153.150
C02506=1090.372,254.692,421.903,176.708,21.007,153.150
C02507=1090.367,254.443,421.930,176.705,21.004,153.150
C02508=1090.360,254.195,421.958,176.702,21.002,153.150
C02509=1090.355,253.946,421.985,176.699,21.000,153.150
C02510=1090.350,253.698,422.013,176.696,20.997,153.150
C02511=1090.344,253.450,422.040,176.693,20.995,153.150
C02512=1090.338,253.200,422.068,176.690,20.993,153.150
C02513=1090.333,252.952,422.094,176.687,20.990,153.150
C02514=1090.327,252.704,422.122,176.684,20.987,153.150
C02515=1090.321,252.456,422.149,176.681,20.985,153.150
C02516=1090.316,252.207,422.176,176.679,20.983,153.150
C02517=1090.310,251.959,422.204,176.676,20.980,153.150
C02518=1090.305,251.710,422.231,176.672,20.978,153.150
C02519=1090.299,251.461,422.258,176.670,20.975,153.149
C02520=1090.294,251.213,422.285,176.667,20.973,153.149
C02521=1090.288,250.964,422.312,176.664,20.970,153.149
C02522=1090.283,250.716,422.340,176.661,20.967,153.149
C02523=1090.277,250.468,422.366,176.658,20.965,153.149
C02524=1090.271,250.220,422.393,176.655,20.963,153.149
C02525=1090.263,249.849,422.434,176.650,20.959,153.149
C02526=1090.255,249.479,422.474,176.647,20.956,153.149
C02527=1090.247,249.108,422.514,176.642,20.952,153.149
C02528=1090.238,248.739,422.554,176.638,20.948,153.149
C02529=1090.233,248.490,422.581,176.635,20.945,153.148
C02530=1090.227,248.242,422.608,176.633,20.944,153.148
C02531=1090.222,247.993,422.635,176.629,20.941,153.148
C02532=1090.217,247.745,422.662,176.626,20.938,153.148
C02533=1090.211,247.496,422.689,176.623,20.936,153.148
C02534=1090.205,247.247,422.716,176.621,20.934,153.148
C02535=1090.199,246.998,422.743,176.618,20.931,153.148
C02536=1090.194,246.750,422.769,176.615,20.928,153.148
C02537=1090.189,246.501,422.797,176.612,20.926,153.148
C02538=1090.183,246.253,422.823,176.609,20.924,153.148
C02539=1090.177,246.005,422.850,176.606,20.922,153.148
C02540=1090.171,245.756,422.876,176.604,20.919,153.148
C02541=1090.166,245.508,422.904,176.600,20.917,153.148
C02542=1090.160,245.259,422.930,176.597,20.914,153.148
C02543=1090.155,245.011,422.957,176.595,20.912,153.148
C02544=1090.149,244.763,422.984,176.592,20.909,153.148
C02545=1090.144,244.513,423.010,176.589,20.907,153.147
C02546=1090.138,244.265,423.037,176.586,20.905,153.147
C02547=1090.133,244.017,423.063,176.583,20.903,153.147
C02548=1090.127,243.768,423.090,176.580,20.900,153.147
C02549=1090.121,243.520,423.117,176.578,20.898,153.147
C02550=1090.115,243.271,423.143,176.574,20.895,153.147
C02551=1090.111,243.022,423.170,176.571,20.893,153.147
C02552=1090.105,242.774,423.197,176.569,20.891,153.147
C02553=1090.099,242.525,423.223,176.566,20.888,153.147
C02554=1090.093,242.277,423.250,176.563,20.886,153.147
C02555=1090.088,242.028,423.276,176.560,20.884,153.147
C02556=1090.082,241.780,423.302,176.557,20.881,153.147
C02557=1090.076,241.531,423.329,176.554,20.879,153.147
C02558=1090.071,241.282,423.355,176.551,20.877,153.147
C02559=1090.065,241.034,423.382,176.548,20.874,153.147
C02560=1090.059,240.786,423.408,176.545,20.871,153.147
C02561=1090.054,240.537,423.434,176.543,20.869,153.147
C02562=1090.048,240.288,423.461,176.540,20.867,153.147
C02563=1090.042,240.040,423.488,176.537,20.865,153.147
C02564=1090.037,239.791,423.513,176.534,20.863,153.147
C02565=1090.031,239.543,423.540,176.531,20.860,153.147
C02566=1090.025,239.294,423.566,176.528,20.858,153.147
C02567=1090.020,239.045,423.593,176.525,20.855,153.146
C02568=1090.014,238.797,423.619,176.522,20.853,153.146
C02569=1090.008,238.548,423.645,176.520,20.851,153.146
C02570=1090.003,238.300,423.672,176.517,20.848,153.146
C02571=1089.996,238.051,423.697,176.513,20.846,153.146
C02572=1089.991,237.803,423.724,176.511,20.844,153.146
C02573=1089.985,237.554,423.750,176.508,20.842,153.146
C02574=1089.980,237.306,423.776,176.506,20.839,153.146
C02575=1089.975,237.057,423.802,176.502,20.837,153.146
C02576=1089.969,236.809,423.829,176.499,20.834,153.146
C02577=1089.960,236.431,423.868,176.495,20.831,153.146
C02578=1089.952,236.054,423.908,176.490,20.827,153.146
C02579=1089.944,235.677,423.947,176.486,20.824,153.146
C02580=1089.935,235.300,423.987,176.482,20.820,153.146
C02581=1089.929,235.051,424.013,176.479,20.818,153.146
C02582=1089.924,234.802,424.039,176.476,20.816,153.146
C02583=1089.918,234.554,424.065,176.474,20.814,153.146
C02584=1089.912,234.305,424.091,176.471,20.811,153.145
C02585=1089.908,234.057,424.117,176.468,20.808,153.145
C02586=1089.901,233.809,424.143,176.465,20.806,153.145
C02587=1089.896,233.560,424.169,176.462,20.804,153.145
C02588=1089.890,233.311,424.195,176.460,20.802,153.145
C02589=1089.884,233.062,424.221,176.456,20.800,153.145
C02590=1089.878,232.814,424.247,176.453,20.797,153.145
C02591=1089.873,232.565,424.272,176.451,20.795,153.145
C02592=1089.868,232.316,424.298,176.448,20.792,153.145
C02593=1089.862,232.067,424.324,176.446,20.790,153.145
C02594=1089.856,231.819,424.350,176.442,20.788,153.145
C02595=1089.851,231.571,424.376,176.439,20.785,153.145
C02596=1089.846,231.322,424.402,176.437,20.783,153.145
C02597=1089.840,231.073,424.428,176.434,20.781,153.145
C02598=1089.834,230.824,424.453,176.431,20.779,153.145
C02599=1089.829,230.576,424.478,176.428,20.776,153.145
C02600=1089.824,230.327,424.504,176.426,20.774,153.145
C02601=1089.817,230.079,424.530,176.423,20.772,153.145
C02602=1089.812,229.830,424.556,176.419,20.769,153.145
C02603=1089.805,229.581,424.582,176.417,20.767,153.145
C02604=1089.800,229.333,424.607,176.414,20.765,153.145
C02605=1089.794,229.084,424.633,176.411,20.763,153.145
C02606=1089.789,228.835,424.659,176.408,20.760,153.145
C02607=1089.783,228.587,424.684,176.406,20.758,153.145
C02608=1089.778,228.339,424.709,176.403,20.756,153.145
C02609=1089.772,228.090,424.735,176.399,20.754,153.145
C02610=1089.766,227.841,424.761,176.397,20.752,153.145
C02611=1089.761,227.592,424.787,176.394,20.749,153.145
C02612=1089.755,227.344,424.812,176.392,20.747,153.144
C02613=1089.749,227.095,424.838,176.388,20.744,153.144
C02614=1089.743,226.846,424.863,176.386,20.742,153.144
C02615=1089.738,226.598,424.888,176.383,20.740,153.144
C02616=1089.732,226.349,424.914,176.381,20.738,153.144
C02617=1089.727,226.100,424.940,176.377,20.735,153.144
C02618=1089.721,225.852,424.964,176.374,20.733,153.144
C02619=1089.716,225.603,424.990,176.372,20.731,153.144
C02620=1089.710,225.354,425.015,176.369,20.729,153.144
C02621=1089.705,225.106,425.041,176.366,20.727,153.144
C02622=1089.699,224.857,425.066,176.363,20.724,153.144
C02623=1089.693,224.608,425.092,176.361,20.722,153.144
C02624=1089.688,224.360,425.117,176.358,20.719,153.144
C02625=1089.682,224.111,425.142,176.355,20.717,153.144
C02626=1089.676,223.862,425.168,176.352,20.715,153.144
C02627=1089.671,223.614,425.193,176.350,20.713,153.144
C02628=1089.665,223.365,425.219,176.346,20.710,153.144
C02629=1089.656,222.979,425.257,176.343,20.707,153.144
C02630=1089.648,222.594,425.296,176.338,20.704,153.144
C02631=1089.639,222.208,425.336,176.334,20.700,153.144
C02632=1089.630,221.822,425.374,176.329,20.696,153.144
C02633=1089.625,221.573,425.400,176.327,20.694,153.144
C02634=1089.619,221.325,425.425,176.324,20.692,153.144
C02635=1089.613,221.076,425.450,176.321,20.690,153.144
C02636=1089.608,220.827,425.476,176.318,20.687,153.144
C02637=1089.603,220.578,425.500,176.316,20.685,153.144
C02638=1089.596,220.330,425.525,176.312,20.683,153.144
C02639=1089.591,220.082,425.550,176.310,20.681,153.144
C02640=1089.585,219.833,425.575,176.307,20.679,153.144
C02641=1089.580,219.584,425.600,176.304,20.677,153.143
C02642=1089.574,219.335,425.625,176.301,20.674,153.143
C02643=1089.568,219.086,425.650,176.299,20.672,153.143
C02644=1089.563,218.838,425.675,176.296,20.670,153.143
C02645=1089.557,218.589,425.701,176.293,20.668,153.143
C02646=1089.552,218.341,425.726,176.290,20.665,153.143
C02647=1089.546,218.091,425.750,176.288,20.663,153.143
C02648=1089.540,217.843,425.774,176.285,20.661,153.143
C02649=1089.534,217.594,425.800,176.282,20.659,153.143
C02650=1089.529,217.346,425.824,176.279,20.656,153.143
C02651=1089.523,217.097,425.850,176.277,20.654,153.143
C02652=1089.518,216.848,425.874,176.274,20.652,153.143
C02653=1089.512,216.599,425.900,176.271,20.650,153.143
C02654=1089.507,216.351,425.924,176.268,20.647,153.143
C02655=1089.500,216.102,425.949,176.266,20.645,153.143
C02656=1089.495,215.854,425.973,176.263,20.643,153.143
C02657=1089.490,215.604,425.999,176.260,20.641,153.143
C02658=1089.484,215.356,426.024,176.257,20.638,153.143
C02659=1089.478,215.107,426.048,176.255,20.636,153.143
C02660=1089.473,214.858,426.072,176.251,20.634,153.143
C02661=1089.468,214.610,426.097,176.249,20.632,153.143
C02662=1089.462,214.361,426.122,176.246,20.630,153.143
C02663=1089.456,214.112,426.146,176.244,20.627,153.143
C02664=1089.450,213.864,426.172,176.241,20.625,153.143
C02665=1089.446,213.615,426.196,176.238,20.623,153.143
C02666=1089.440,213.366,426.221,176.235,20.620,153.143
C02667=1089.434,213.117,426.245,176.233,20.618,153.143
C02668=1089.429,212.869,426.270,176.229,20.616,153.143
C02669=1089.423,212.620,426.295,176.227,20.614,153.143
C02670=1089.418,212.371,426.319,176.224,20.611,153.143
C02671=1089.412,212.122,426.344,176.221,20.609,153.143
C02672=1089.406,211.874,426.369,176.219,20.607,153.143
C02673=1089.401,211.625,426.393,176.216,20.605,153.143
C02674=1089.395,211.376,426.418,176.214,20.603,153.142
C02675=1089.390,211.127,426.442,176.210,20.601,153.142
C02676=1089.383,210.878,426.466,176.208,20.599,153.142
C02677=1089.378,210.630,426.490,176.205,20.596,153.142
C02678=1089.372,210.381,426.514,176.202,20.594,153.142
C02679=1089.366,210.132,426.540,176.199,20.592,153.142
C02680=1089.361,209.884,426.564,176.197,20.590,153.142
C02681=1089.352,209.502,426.602,176.193,20.586,153.142
C02682=1089.344,209.120,426.638,176.188,20.582,153.142
C02683=1089.335,208.738,426.676,176.184,20.579,153.142
C02684=1089.326,208.356,426.714,176.180,20.576,153.142
C02685=1089.303,207.333,426.812,176.110,20.541,153.146
C02686=1089.298,207.084,426.836,176.107,20.540,153.146
C02687=1089.293,206.836,426.860,176.104,20.539,153.147
C02688=1089.287,206.587,426.884,176.101,20.537,153.147
C02689=1089.282,206.338,426.907,176.098,20.536,153.147
C02690=1089.276,206.089,426.932,176.096,20.534,153.147
C02691=1089.270,205.841,426.955,176.093,20.533,153.147
C02692=1089.265,205.591,426.979,176.090,20.532,153.147
C02693=1089.259,205.343,427.003,176.088,20.531,153.148
C02694=1089.253,205.094,427.027,176.084,20.529,153.148
C02695=1089.248,204.845,427.050,176.081,20.528,153.148
C02696=1089.242,204.596,427.075,176.078,20.527,153.148
C02697=1089.236,204.348,427.099,176.076,20.525,153.148
C02698=1089.231,204.099,427.122,176.073,20.524,153.149
C02699=1089.225,203.850,427.146,176.071,20.523,153.149
C02700=1089.220,203.601,427.170,176.067,20.521,153.149
C02701=1089.214,203.353,427.193,176.064,20.520,153.149
C02702=1089.209,203.104,427.217,176.062,20.518,153.149
C02703=1089.203,202.855,427.240,176.059,20.517,153.150
C02704=1089.198,202.605,427.264,176.056,20.516,153.150
C02705=1089.192,202.357,427.288,176.054,20.515,153.150
C02706=1089.187,202.108,427.311,176.050,20.513,153.150
C02707=1089.181,201.860,427.335,176.047,20.512,153.150
C02708=1089.175,201.611,427.358,176.045,20.511,153.151
C02709=1089.170,201.362,427.382,176.042,20.510,153.151
C02710=1089.164,201.113,427.405,176.039,20.509,153.151
C02711=1089.158,200.864,427.430,176.036,20.508,153.151
C02712=1089.152,200.615,427.453,176.034,20.506,153.151
C02713=1089.146,200.367,427.477,176.030,20.505,153.152
C02714=1089.141,200.118,427.500,176.028,20.503,153.152
C02715=1089.135,199.869,427.523,176.025,20.502,153.152
C02716=1089.129,199.620,427.547,176.022,20.501,153.152
C02717=1089.124,199.371,427.570,176.019,20.500,153.152
C02718=1089.118,199.123,427.594,176.017,20.499,153.153
C02719=1089.113,198.874,427.617,176.014,20.497,153.153
C02720=1089.107,198.624,427.641,176.011,20.496,153.153
C02721=1089.101,198.376,427.664,176.008,20.494,153.153
C02722=1089.095,198.127,427.687,176.005,20.493,153.153
C02723=1089.090,197.878,427.711,176.003,20.492,153.153
C02724=1089.084,197.629,427.735,176.000,20.491,153.154
C02725=1089.079,197.381,427.757,175.997,20.489,153.154
C02726=1089.073,197.132,427.780,175.994,20.488,153.154
C02727=1089.068,196.882,427.804,175.992,20.487,153.154
C02728=1089.062,196.634,427.828,175.989,20.486,153.154
C02729=1089.056,196.385,427.851,175.986,20.484,153.154
C02730=1089.051,196.136,427.874,175.983,20.483,153.155
C02731=1089.045,195.887,427.897,175.980,20.481,153.155
C02732=1089.039,195.639,427.921,175.977,20.480,153.155
C02733=1089.034,195.390,427.944,175.975,20.479,153.155
C02734=1089.029,195.141,427.967,175.972,20.478,153.155
C02735=1089.023,194.892,427.990,175.969,20.477,153.156
C02736=1089.017,194.643,428.013,175.967,20.476,153.156
C02737=1089.011,194.394,428.036,175.964,20.474,153.156
C02738=1089.006,194.145,428.060,175.962,20.473,153.156
C02739=1089.000,193.897,428.083,175.959,20.472,153.156
C02740=1088.995,193.648,428.106,175.956,20.470,153.156
C02741=1088.989,193.399,428.129,175.953,20.469,153.157
C02742=1088.984,193.150,428.153,175.950,20.467,153.157
C02743=1088.978,192.901,428.176,175.947,20.466,153.157
C02744=1088.973,192.652,428.198,175.945,20.465,153.157
C02745=1088.967,192.404,428.221,175.942,20.463,153.157
C02746=1088.960,192.126,428.247,175.939,20.462,153.158
C02747=1088.955,191.849,428.273,175.936,20.460,153.158
C02748=1088.949,191.572,428.298,175.933,20.459,153.158
C02749=1088.942,191.295,428.325,175.930,20.457,153.158
C02750=1088.936,191.046,428.347,175.927,20.456,153.158
C02751=1088.931,190.797,428.370,175.924,20.455,153.158
C02752=1088.926,190.549,428.394,175.922,20.453,153.159
C02753=1088.921,190.300,428.417,175.919,20.452,153.159
C02754=1088.915,190.051,428.439,175.916,20.451,153.159
C02755=1088.909,189.802,428.462,175.914,20.450,153.159
C02756=1088.903,189.553,428.485,175.911,20.449,153.159
C02757=1088.898,189.304,428.508,175.908,20.447,153.159
C02758=1088.893,189.054,428.531,175.906,20.446,153.160
C02759=1088.888,188.806,428.554,175.903,20.445,153.160
C02760=1088.882,188.557,428.577,175.900,20.443,153.160
C02761=1088.876,188.308,428.600,175.898,20.442,153.160
C02762=1088.871,188.059,428.623,175.895,20.441,153.160
C02763=1088.865,187.811,428.645,175.892,20.439,153.160
C02764=1088.860,187.562,428.668,175.890,20.438,153.161
C02765=1088.855,187.313,428.692,175.886,20.436,153.161
C02766=1088.849,187.064,428.714,175.884,20.435,153.161
C02767=1088.844,186.815,428.737,175.881,20.433,153.161
C02768=1088.838,186.566,428.760,175.878,20.432,153.161
C02769=1088.833,186.318,428.782,175.876,20.431,153.161
C02770=1088.827,186.069,428.805,175.873,20.429,153.162
C02771=1088.822,185.819,428.827,175.871,20.428,153.162
C02772=1088.816,185.570,428.850,175.868,20.427,153.162
C02773=1088.811,185.322,428.873,175.865,20.425,153.162
C02774=1088.805,185.073,428.896,175.863,20.424,153.162
C02775=1088.800,184.824,428.918,175.860,20.423,153.162
C02776=1088.794,184.575,428.941,175.857,20.422,153.162
C02777=1088.788,184.326,428.964,175.854,20.421,153.163
C02778=1088.783,184.076,428.986,175.852,20.419,153.163
C02779=1088.776,183.828,429.009,175.849,20.418,153.163
C02780=1088.771,183.580,429.031,175.847,20.417,153.163
C02781=1088.766,183.330,429.053,175.844,20.416,153.163
C02782=1088.760,183.081,429.076,175.841,20.414,153.164
C02783=1088.754,182.833,429.099,175.838,20.413,153.164
C02784=1088.748,182.583,429.121,175.836,20.412,153.164
C02785=1088.742,182.334,429.144,175.833,20.410,153.164
C02786=1088.737,182.086,429.166,175.830,20.409,153.164
C02787=1088.731,181.837,429.188,175.828,20.408,153.164
C02788=1088.725,181.588,429.211,175.825,20.407,153.165
C02789=1088.720,181.338,429.233,175.823,20.405,153.165
C02790=1088.713,181.090,429.256,175.820,20.404,153.165
C02791=1088.708,180.841,429.279,175.817,20.403,153.165
C02792=1088.703,180.592,429.300,175.815,20.401,153.165
C02793=1088.696,180.344,429.323,175.812,20.400,153.166
C02794=1088.691,180.094,429.345,175.809,20.399,153.166
C02795=1088.685,179.845,429.368,175.806,20.398,153.166
C02796=1088.680,179.596,429.390,175.804,20.396,153.166
C02797=1088.674,179.348,429.412,175.801,20.395,153.166
C02798=1088.669,179.098,429.434,175.798,20.394,153.166
C02799=1088.663,178.849,429.457,175.796,20.393,153.167
C02800=1088.657,178.601,429.479,175.793,20.391,153.167
C02801=1088.652,178.352,429.502,175.791,20.390,153.167
C02802=1088.646,178.102,429.524,175.788,20.389,153.167
C02803=1088.640,177.854,429.546,175.785,20.387,153.167
C02804=1088.635,177.605,429.568,175.783,20.386,153.167
C02805=1088.629,177.356,429.590,175.780,20.385,153.168
C02806=1088.623,177.107,429.613,175.777,20.383,153.168
C02807=1088.618,176.858,429.635,175.775,20.382,153.168
C02808=1088.612,176.609,429.657,175.772,20.381,153.168
C02809=1088.606,176.360,429.679,175.770,20.379,153.168
C02810=1088.601,176.082,429.704,175.767,20.378,153.168
C02811=1088.594,175.806,429.728,175.764,20.377,153.168
C02812=1088.588,175.527,429.753,175.761,20.375,153.169
C02813=1088.582,175.250,429.778,175.758,20.374,153.169
C02814=1088.576,175.002,429.799,175.755,20.372,153.169
C02815=1088.571,174.752,429.822,175.753,20.371,153.169
C02816=1088.564,174.504,429.844,175.750,20.369,153.169
C02817=1088.559,174.255,429.866,175.747,20.369,153.170
C02818=1088.554,174.005,429.888,175.745,20.367,153.170
C02819=1088.548,173.756,429.910,175.742,20.366,153.170
C02820=1088.543,173.508,429.932,175.740,20.364,153.170
C02821=1088.536,173.259,429.954,175.737,20.363,153.170
C02822=1088.532,173.010,429.976,175.734,20.362,153.170
C02823=1088.525,172.761,429.997,175.733,20.361,153.170
C02824=1088.520,172.512,430.020,175.730,20.359,153.170
C02825=1088.515,172.263,430.042,175.727,20.358,153.171
C02826=1088.509,172.014,430.064,175.725,20.357,153.171
C02827=1088.504,171.765,430.086,175.722,20.355,153.171
C02828=1088.498,171.516,430.107,175.720,20.354,153.171
C02829=1088.492,171.266,430.130,175.717,20.352,153.171
C02830=1088.486,171.018,430.151,175.714,20.351,153.171
C02831=1088.481,170.769,430.174,175.712,20.350,153.172
C02832=1088.475,170.520,430.195,175.709,20.348,153.172
C02833=1088.470,170.271,430.217,175.706,20.347,153.172
C02834=1088.464,170.022,430.238,175.704,20.345,153.172
C02835=1088.459,169.773,430.261,175.701,20.344,153.172
C02836=1088.453,169.524,430.282,175.699,20.342,153.172
C02837=1088.448,169.275,430.304,175.696,20.341,153.172
C02838=1088.443,169.026,430.326,175.693,20.340,153.173
C02839=1088.437,168.777,430.348,175.692,20.339,153.173
C02840=1088.432,168.528,430.370,175.689,20.338,153.173
C02841=1088.426,168.279,430.391,175.687,20.336,153.173
C02842=1088.420,168.030,430.412,175.684,20.335,153.173
C02843=1088.415,167.781,430.435,175.681,20.333,153.173
C02844=1088.409,167.532,430.456,175.679,20.332,153.173
C02845=1088.404,167.283,430.478,175.676,20.330,153.173
C02846=1088.398,167.034,430.499,175.674,20.329,153.173
C02847=1088.393,166.785,430.522,175.671,20.327,153.174
C02848=1088.387,166.536,430.543,175.669,20.326,153.174
C02849=1088.382,166.287,430.565,175.666,20.324,153.174
C02850=1088.376,166.038,430.586,175.663,20.323,153.174
C02851=1088.372,165.789,430.608,175.661,20.322,153.174
C02852=1088.366,165.540,430.630,175.659,20.321,153.174
C02853=1088.361,165.291,430.652,175.656,20.319,153.174
C02854=1088.355,165.042,430.673,175.654,20.318,153.174
C02855=1088.349,164.793,430.695,175.651,20.316,153.175
C02856=1088.344,164.544,430.717,175.649,20.315,153.175
C02857=1088.338,164.295,430.738,175.646,20.314,153.175
C02858=1088.333,164.046,430.759,175.644,20.312,153.175
C02859=1088.327,163.797,430.781,175.641,20.311,153.175
C02860=1088.322,163.548,430.803,175.638,20.309,153.175
C02861=1088.316,163.299,430.825,175.637,20.308,153.175
C02862=1088.311,163.050,430.845,175.634,20.307,153.175
C02863=1088.306,162.801,430.867,175.632,20.305,153.176
C02864=1088.300,162.552,430.889,175.629,20.304,153.176
C02865=1088.295,162.303,430.910,175.626,20.302,153.176
C02866=1088.290,162.054,430.932,175.624,20.301,153.176
C02867=1088.284,161.805,430.953,175.621,20.299,153.176
C02868=1088.279,161.556,430.975,175.619,20.297,153.176
C02869=1088.273,161.307,430.996,175.616,20.296,153.176
C02870=1088.267,161.058,431.017,175.614,20.295,153.176
C02871=1088.262,160.809,431.038,175.612,20.294,153.176
C02872=1088.256,160.560,431.060,175.609,20.292,153.177
C02873=1088.250,160.311,431.081,175.607,20.291,153.177
C02874=1088.245,160.033,431.105,175.604,20.289,153.177
C02875=1088.238,159.755,431.129,175.602,20.288,153.177
C02876=1088.232,159.477,431.152,175.598,20.286,153.177
C02877=1088.225,159.199,431.176,175.596,20.285,153.177
C02878=1088.220,158.951,431.197,175.593,20.283,153.177
C02879=1088.214,158.701,431.218,175.590,20.282,153.177
C02880=1088.209,158.452,431.240,175.589,20.281,153.178
C02881=1088.204,158.203,431.260,175.586,20.279,153.178
C02882=1088.198,157.954,431.282,175.584,20.278,153.178
C02883=1088.192,157.706,431.303,175.581,20.276,153.178
C02884=1088.187,157.456,431.324,175.578,20.275,153.178
C02885=1088.181,157.207,431.345,175.576,20.273,153.178
C02886=1088.175,156.958,431.366,175.573,20.272,153.178
C02887=1088.170,156.710,431.387,175.572,20.271,153.178
C02888=1088.164,156.460,431.408,175.569,20.269,153.178
C02889=1088.158,156.211,431.429,175.566,20.268,153.179
C02890=1088.153,155.962,431.450,175.564,20.266,153.179
C02891=1088.148,155.713,431.472,175.561,20.265,153.179
C02892=1088.143,155.463,431.493,175.559,20.263,153.179
C02893=1088.137,155.215,431.514,175.556,20.262,153.179
C02894=1088.130,154.965,431.534,175.554,20.261,153.179
C02895=1088.125,154.717,431.556,175.552,20.260,153.179
C02896=1088.120,154.468,431.576,175.549,20.258,153.179
C02897=1088.113,154.219,431.598,175.547,20.257,153.180
C02898=1088.108,153.969,431.618,175.544,20.255,153.180
C02899=1088.103,153.721,431.640,175.542,20.254,153.180
C02900=1088.097,153.471,431.661,175.540,20.253,153.180
C02901=1088.091,153.223,431.682,175.537,20.251,153.180
C02902=1088.086,152.974,431.702,175.535,20.250,153.180
C02903=1088.080,152.724,431.723,175.532,20.248,153.180
C02904=1088.074,152.475,431.745,175.530,20.247,153.180
C02905=1088.069,152.226,431.765,175.527,20.245,153.180
C02906=1088.064,151.977,431.786,175.525,20.244,153.181
C02907=1088.058,151.728,431.807,175.523,20.243,153.181
C02908=1088.053,151.479,431.828,175.520,20.241,153.181
C02909=1088.047,151.229,431.848,175.518,20.239,153.181
C02910=1088.042,150.981,431.870,175.515,20.238,153.181
C02911=1088.035,150.731,431.890,175.513,20.236,153.181
C02912=1088.030,150.482,431.911,175.511,20.235,153.181
C02913=1088.024,150.234,431.932,175.508,20.234,153.181
C02914=1088.019,149.985,431.952,175.506,20.233,153.181
C02915=1088.014,149.736,431.973,175.503,20.231,153.181
C02916=1088.008,149.486,431.994,175.501,20.230,153.182
C02917=1088.002,149.237,432.015,175.499,20.229,153.182
C02918=1087.997,148.988,432.036,175.497,20.227,153.182
C02919=1087.991,148.739,432.056,175.494,20.225,153.182
C02920=1087.985,148.489,432.077,175.492,20.224,153.182
C02921=1087.980,148.241,432.098,175.489,20.222,153.182
C02922=1087.974,147.992,432.118,175.487,20.221,153.182
C02923=1087.968,147.743,432.138,175.485,20.220,153.182
C02924=1087.963,147.494,432.159,175.482,20.218,153.182
C02925=1087.957,147.244,432.180,175.480,20.217,153.182
C02926=1087.952,146.995,432.200,175.477,20.215,153.183
C02927=1087.946,146.747,432.221,175.475,20.214,153.183
C02928=1087.941,146.498,432.242,175.473,20.212,153.183
C02929=1087.935,146.249,432.262,175.470,20.211,153.183
C02930=1087.929,145.999,432.283,175.468,20.209,153.183
C02931=1087.923,145.750,432.303,175.465,20.208,153.183
C02932=1087.918,145.501,432.324,175.464,20.207,153.183
C02933=1087.913,145.252,432.344,175.461,20.205,153.183
C02934=1087.907,145.003,432.364,175.459,20.204,153.183
C02935=1087.901,144.753,432.385,175.456,20.202,153.183
C02936=1087.896,144.505,432.406,175.453,20.201,153.183
C02937=1087.890,144.256,432.426,175.452,20.200,153.184
C02938=1087.884,143.977,432.449,175.449,20.198,153.184
C02939=1087.878,143.699,432.472,175.446,20.196,153.184
C02940=1087.871,143.421,432.495,175.443,20.194,153.184
C02941=1087.865,143.143,432.517,175.441,20.193,153.184
C02942=1087.859,142.894,432.538,175.438,20.191,153.184
C02943=1087.854,142.645,432.559,175.437,20.190,153.184
C02944=1087.848,142.396,432.579,175.434,20.188,153.184
C02945=1087.843,142.147,432.599,175.432,20.187,153.184
C02946=1087.838,141.898,432.620,175.429,20.185,153.184
C02947=1087.831,141.648,432.639,175.427,20.184,153.184
C02948=1087.826,141.399,432.660,175.425,20.182,153.184
C02949=1087.820,141.150,432.680,175.422,20.181,153.185
C02950=1087.815,140.901,432.700,175.420,20.179,153.185
C02951=1087.810,140.652,432.721,175.418,20.178,153.185
C02952=1087.804,140.403,432.741,175.416,20.176,153.185
C02953=1087.798,140.154,432.761,175.413,20.175,153.185
C02954=1087.792,139.905,432.781,175.411,20.174,153.185
C02955=1087.787,139.656,432.802,175.408,20.172,153.185
C02956=1087.781,139.407,432.822,175.407,20.171,153.185
C02957=1087.776,139.157,432.842,175.404,20.169,153.185
C02958=1087.770,138.909,432.862,175.402,20.168,153.185
C02959=1087.764,138.659,432.883,175.399,20.166,153.185
C02960=1087.758,138.410,432.903,175.397,20.165,153.185
C02961=1087.753,138.161,432.923,175.395,20.163,153.186
C02962=1087.747,137.912,432.943,175.392,20.162,153.186
C02963=1087.742,137.662,432.963,175.390,20.160,153.186
C02964=1087.736,137.413,432.983,175.388,20.159,153.186
C02965=1087.731,137.164,433.003,175.386,20.157,153.186
C02966=1087.725,136.916,433.023,175.383,20.156,153.186
C02967=1087.720,136.666,433.043,175.381,20.154,153.186
C02968=1087.714,136.417,433.063,175.379,20.153,153.186
C02969=1087.708,136.168,433.083,175.377,20.151,153.186
C02970=1087.703,135.919,433.104,175.374,20.149,153.186
C02971=1087.697,135.670,433.123,175.372,20.148,153.186
C02972=1087.692,135.420,433.143,175.370,20.147,153.186
C02973=1087.686,135.172,433.163,175.368,20.145,153.186
C02974=1087.681,134.922,433.183,175.365,20.144,153.187
C02975=1087.675,134.673,433.203,175.363,20.143,153.187
C02976=1087.669,134.424,433.223,175.361,20.141,153.187
C02977=1087.664,134.175,433.243,175.358,20.139,153.187
C02978=1087.658,133.926,433.263,175.356,20.138,153.187
C02979=1087.653,133.677,433.284,175.354,20.136,153.187
C02980=1087.647,133.427,433.303,175.352,20.135,153.187
C02981=1087.641,133.178,433.323,175.349,20.133,153.187
C02982=1087.636,132.929,433.343,175.347,20.131,153.187
C02983=1087.630,132.680,433.363,175.345,20.130,153.187
C02984=1087.624,132.431,433.383,175.343,20.128,153.187
C02985=1087.619,132.181,433.402,175.340,20.127,153.187
C02986=1087.613,131.932,433.422,175.339,20.126,153.187
C02987=1087.607,131.683,433.442,175.336,20.124,153.187
C02988=1087.601,131.434,433.462,175.334,20.122,153.187
C02989=1087.596,131.185,433.482,175.331,20.121,153.188
C02990=1087.590,130.936,433.501,175.330,20.119,153.187
C02991=1087.584,130.687,433.521,175.327,20.118,153.188
C02992=1087.579,130.437,433.541,175.324,20.116,153.188
C02993=1087.573,130.189,433.560,175.323,20.115,153.188
C02994=1087.567,129.939,433.580,175.320,20.113,153.188
C02995=1087.562,129.690,433.600,175.318,20.112,153.188
C02996=1087.556,129.441,433.620,175.316,20.110,153.188
C02997=1087.550,129.192,433.639,175.314,20.109,153.188
C02998=1087.544,128.942,433.659,175.311,20.108,153.188
C02999=1087.539,128.693,433.678,175.309,20.106,153.188
C03000=1087.533,128.444,433.698,175.307,20.105,153.188
C03001=1087.528,128.195,433.717,175.305,20.103,153.188
C03002=1087.522,127.917,433.739,175.302,20.101,153.188
C03003=1087.515,127.638,433.761,175.300,20.099,153.188
C03004=1087.508,127.361,433.784,175.297,20.098,153.188
C03005=1087.502,127.083,433.805,175.295,20.096,153.189
C03006=1087.496,126.833,433.825,175.292,20.094,153.189
C03007=1087.491,126.584,433.843,175.290,20.093,153.189
C03008=1087.485,126.336,433.863,175.288,20.091,153.189
C03009=1087.479,126.086,433.883,175.286,20.090,153.189
C03010=1087.474,125.837,433.902,175.284,20.088,153.189
C03011=1087.468,125.588,433.922,175.282,20.087,153.189
C03012=1087.463,125.338,433.942,175.279,20.085,153.189
C03013=1087.457,125.089,433.961,175.277,20.083,153.189
C03014=1087.451,124.840,433.981,175.275,20.082,153.189
C03015=1087.446,124.591,434.000,175.273,20.080,153.189
C03016=1087.440,124.342,434.019,175.271,20.079,153.189
C03017=1087.435,124.092,434.038,175.269,20.078,153.189
C03018=1087.429,123.843,434.058,175.267,20.076,153.189
C03019=1087.423,123.594,434.077,175.264,20.074,153.189
C03020=1087.417,123.345,434.097,175.262,20.072,153.189
C03021=1087.412,123.095,434.116,175.260,20.071,153.189
C03022=1087.406,122.847,434.136,175.258,20.069,153.189
C03023=1087.400,122.598,434.155,175.255,20.068,153.189
C03024=1087.395,122.348,434.174,175.254,20.066,153.189
C03025=1087.390,122.098,434.194,175.251,20.065,153.189
C03026=1087.384,121.850,434.214,175.249,20.063,153.189
C03027=1087.379,121.601,434.233,175.247,20.062,153.190
C03028=1087.373,121.351,434.252,175.245,20.060,153.190
C03029=1087.367,121.102,434.271,175.242,20.058,153.190
C03030=1087.362,120.853,434.290,175.241,20.057,153.190
C03031=1087.356,120.603,434.310,175.238,20.055,153.190
C03032=1087.351,120.354,434.329,175.236,20.053,153.190
C03033=1087.345,120.106,434.349,175.234,20.052,153.190
C03034=1087.339,119.856,434.368,175.232,20.050,153.190
C03035=1087.334,119.607,434.387,175.229,20.048,153.190
C03036=1087.328,119.358,434.406,175.228,20.047,153.190
C03037=1087.323,119.109,434.425,175.225,20.045,153.190
C03038=1087.317,118.859,434.444,175.223,20.043,153.190
C03039=1087.311,118.610,434.464,175.221,20.042,153.190
C03040=1087.306,118.361,434.483,175.219,20.041,153.190
C03041=1087.301,118.112,434.502,175.216,20.039,153.190
C03042=1087.295,117.862,434.521,175.215,20.037,153.190
C03043=1087.290,117.613,434.540,175.212,20.036,153.190
C03044=1087.284,117.364,434.559,175.210,20.034,153.190
C03045=1087.278,117.115,434.578,175.209,20.032,153.190
C03046=1087.273,116.866,434.597,175.206,20.031,153.190
C03047=1087.267,116.617,434.616,175.204,20.029,153.190
C03048=1087.261,116.367,434.635,175.202,20.027,153.190
C03049=1087.256,116.118,434.654,175.200,20.025,153.190
C03050=1087.250,115.869,434.673,175.197,20.024,153.190
C03051=1087.245,115.620,434.692,175.196,20.022,153.190
C03052=1087.239,115.370,434.712,175.194,20.020,153.190
C03053=1087.234,115.121,434.731,175.192,20.019,153.190
C03054=1087.228,114.872,434.750,175.189,20.017,153.190
C03055=1087.223,114.623,434.769,175.187,20.015,153.190
C03056=1087.218,114.374,434.788,175.186,20.014,153.190
C03057=1087.212,114.124,434.807,175.183,20.012,153.190
C03058=1087.205,113.875,434.826,175.181,20.010,153.190
C03059=1087.201,113.626,434.844,175.179,20.009,153.190
C03060=1087.195,113.377,434.863,175.177,20.007,153.190
C03061=1087.189,113.127,434.883,175.174,20.005,153.190
C03062=1087.183,112.879,434.901,175.173,20.004,153.190
C03063=1087.178,112.629,434.920,175.170,20.002,153.190
C03064=1087.172,112.380,434.939,175.168,20.000,153.190
C03065=1087.167,112.131,434.958,175.167,19.999,153.190
C03066=1087.160,111.853,434.979,175.164,19.997,153.190
C03067=1087.154,111.574,434.999,175.162,19.996,153.190
C03068=1087.148,111.296,435.021,175.159,19.994,153.190
C03069=1087.141,111.018,435.041,175.157,19.992,153.190
C03070=1087.136,110.769,435.061,175.155,19.990,153.190
C03071=1087.130,110.519,435.080,175.153,19.989,153.190
C03072=1087.125,110.270,435.097,175.151,19.987,153.190
C03073=1087.119,110.021,435.117,175.149,19.985,153.190
C03074=1087.112,109.772,435.135,175.147,19.984,153.191
C03075=1087.107,109.523,435.154,175.144,19.982,153.191
C03076=1087.102,109.273,435.173,175.143,19.980,153.190
C03077=1087.096,109.024,435.191,175.140,19.978,153.190
C03078=1087.090,108.775,435.210,175.139,19.977,153.191
C03079=1087.085,108.526,435.229,175.136,19.975,153.191
C03080=1087.079,108.277,435.247,175.134,19.973,153.191
C03081=1087.074,108.027,435.266,175.132,19.972,153.191
C03082=1087.067,107.778,435.285,175.130,19.970,153.191
C03083=1087.062,107.529,435.303,175.128,19.968,153.191
C03084=1087.057,107.279,435.322,175.126,19.967,153.191
C03085=1087.051,107.031,435.341,175.124,19.965,153.191
C03086=1087.045,106.781,435.359,175.122,19.964,153.191
C03087=1087.039,106.532,435.378,175.120,19.962,153.191
C03088=1087.034,106.282,435.396,175.117,19.960,153.191
C03089=1087.028,106.033,435.415,175.116,19.958,153.191
C03090=1087.023,105.784,435.433,175.114,19.956,153.191
C03091=1087.017,105.534,435.452,175.112,19.955,153.191
C03092=1087.011,105.285,435.471,175.110,19.953,153.191
C03093=1087.006,105.036,435.489,175.107,19.951,153.191
C03094=1087.000,104.787,435.507,175.106,19.950,153.191
C03095=1086.995,104.537,435.526,175.103,19.948,153.191
C03096=1086.988,104.288,435.544,175.102,19.947,153.191
C03097=1086.984,104.039,435.562,175.099,19.945,153.191
C03098=1086.977,103.790,435.581,175.097,19.943,153.191
C03099=1086.972,103.541,435.600,175.096,19.942,153.191
C03100=1086.966,103.291,435.618,175.093,19.940,153.191
C03101=1086.961,103.043,435.637,175.092,19.938,153.191
C03102=1086.955,102.793,435.655,175.090,19.936,153.191
C03103=1086.950,102.544,435.673,175.087,19.934,153.191
C03104=1086.944,102.294,435.692,175.085,19.933,153.191
C03105=1086.939,102.045,435.710,175.083,19.931,153.191
C03106=1086.932,101.796,435.728,175.082,19.930,153.191
C03107=1086.928,101.547,435.746,175.079,19.928,153.191
C03108=1086.921,101.297,435.765,175.077,19.926,153.191
C03109=1086.916,101.048,435.783,175.076,19.924,153.191
C03110=1086.910,100.799,435.802,175.073,19.922,153.190
C03111=1086.905,100.550,435.820,175.072,19.921,153.190
C03112=1086.899,100.300,435.838,175.069,19.919,153.191
C03113=1086.893,100.051,435.856,175.068,19.918,153.191
C03114=1086.888,99.801,435.875,175.065,19.916,153.191
C03115=1086.882,99.553,435.893,175.063,19.914,153.191
C03116=1086.876,99.303,435.911,175.062,19.912,153.190
C03117=1086.871,99.054,435.929,175.059,19.910,153.190
C03118=1086.865,98.805,435.948,175.058,19.909,153.190
C03119=1086.859,98.556,435.965,175.055,19.907,153.191
C03120=1086.853,98.306,435.983,175.053,19.905,153.191
C03121=1086.848,98.057,436.002,175.051,19.904,153.190
C03122=1086.842,97.808,436.020,175.049,19.902,153.190
C03123=1086.836,97.558,436.038,175.048,19.900,153.190
C03124=1086.831,97.308,436.056,175.045,19.898,153.190
C03125=1086.825,97.060,436.075,175.044,19.897,153.190
C03126=1086.819,96.810,436.093,175.041,19.895,153.190
C03127=1086.814,96.561,436.111,175.039,19.893,153.190
C03128=1086.808,96.312,436.129,175.038,19.891,153.190
C03129=1086.802,96.063,436.147,175.035,19.889,153.190
C03130=1086.796,95.785,436.167,175.033,19.887,153.190
C03131=1086.790,95.506,436.186,175.031,19.886,153.190
C03132=1086.784,95.228,436.207,175.029,19.884,153.190
C03133=1086.777,94.950,436.228,175.027,19.882,153.190
C03134=1086.772,94.701,436.245,175.024,19.880,153.190
C03135=1086.766,94.451,436.263,175.023,19.879,153.190
C03136=1086.760,94.202,436.281,175.021,19.877,153.190
C03137=1086.755,93.953,436.300,175.019,19.875,153.190
C03138=1086.749,93.703,436.318,175.017,19.873,153.190
C03139=1086.743,93.454,436.335,175.015,19.872,153.190
C03140=1086.738,93.205,436.353,175.013,19.870,153.190
C03141=1086.732,92.955,436.371,175.011,19.868,153.190
C03142=1086.727,92.707,436.389,175.009,19.866,153.190
C03143=1086.721,92.458,436.407,175.007,19.864,153.190
C03144=1086.715,92.208,436.425,175.005,19.863,153.190
C03145=1086.710,91.959,436.443,175.003,19.861,153.190
C03146=1086.705,91.710,436.461,175.002,19.859,153.190
C03147=1086.699,91.460,436.479,174.999,19.857,153.190
C03148=1086.693,91.211,436.496,174.998,19.856,153.190
C03149=1086.687,90.961,436.514,174.996,19.854,153.190
C03150=1086.681,90.712,436.532,174.993,19.852,153.190
C03151=1086.676,90.463,436.549,174.992,19.850,153.190
C03152=1086.671,90.213,436.568,174.989,19.848,153.190
C03153=1086.665,89.964,436.585,174.988,19.847,153.190
C03154=1086.659,89.715,436.603,174.986,19.845,153.190
C03155=1086.653,89.465,436.621,174.984,19.843,153.190
C03156=1086.648,89.216,436.638,174.982,19.841,153.190
C03157=1086.642,88.966,436.656,174.980,19.840,153.190
C03158=1086.636,88.717,436.674,174.978,19.838,153.190
C03159=1086.631,88.468,436.692,174.977,19.836,153.190
C03160=1086.625,88.218,436.709,174.974,19.834,153.190
C03161=1086.619,87.969,436.727,174.972,19.832,153.190
C03162=1086.614,87.720,436.745,174.970,19.831,153.189
C03163=1086.607,87.471,436.763,174.968,19.829,153.189
C03164=1086.602,87.222,436.780,174.967,19.827,153.189
C03165=1086.596,86.973,436.798,174.964,19.825,153.189
C03166=1086.590,86.723,436.816,174.963,19.824,153.189
C03167=1086.585,86.474,436.833,174.961,19.821,153.189
C03168=1086.579,86.225,436.851,174.959,19.820,153.189
C03169=1086.573,85.975,436.869,174.957,19.818,153.189
C03170=1086.568,85.726,436.886,174.955,19.816,153.189
C03171=1086.562,85.476,436.903,174.953,19.814,153.189
C03172=1086.556,85.227,436.921,174.952,19.813,153.189
C03173=1086.551,84.978,436.939,174.949,19.811,153.189
C03174=1086.545,84.728,436.956,174.948,19.809,153.189
C03175=1086.539,84.480,436.973,174.946,19.807,153.189
C03176=1086.533,84.230,436.991,174.944,19.806,153.189
C03177=1086.527,83.981,437.009,174.942,19.804,153.189
C03178=1086.522,83.731,437.025,174.940,19.802,153.189
C03179=1086.517,83.482,437.043,174.938,19.800,153.189
C03180=1086.510,83.233,437.061,174.936,19.798,153.189
C03181=1086.505,82.983,437.079,174.934,19.796,153.189
C03182=1086.499,82.734,437.096,174.932,19.794,153.189
C03183=1086.494,82.485,437.113,174.931,19.793,153.189
C03184=1086.488,82.235,437.131,174.928,19.791,153.189
C03185=1086.483,81.986,437.148,174.927,19.789,153.188
C03186=1086.477,81.737,437.166,174.925,19.787,153.188
C03187=1086.472,81.487,437.183,174.923,19.786,153.188
C03188=1086.466,81.238,437.201,174.921,19.784,153.188
C03189=1086.460,80.989,437.218,174.919,19.782,153.188
C03190=1086.454,80.739,437.235,174.917,19.780,153.188
C03191=1086.449,80.490,437.252,174.916,19.778,153.188
C03192=1086.443,80.241,437.270,174.914,19.776,153.188
C03193=1086.438,79.991,437.287,174.912,19.775,153.188
C03194=1086.432,79.714,437.307,174.910,19.773,153.188
C03195=1086.425,79.435,437.326,174.908,19.770,153.188
C03196=1086.419,79.157,437.345,174.905,19.768,153.188
C03197=1086.413,78.878,437.364,174.904,19.766,153.188
C03198=1086.407,78.629,437.382,174.902,19.764,153.188
C03199=1086.401,78.381,437.399,174.900,19.763,153.188
C03200=1086.396,78.131,437.416,174.898,19.761,153.188
C03201=1086.390,77.882,437.433,174.896,19.759,153.188
C03202=1086.385,77.633,437.451,174.894,19.757,153.188
C03203=1086.378,77.383,437.468,174.893,19.755,153.187
C03204=1086.373,77.134,437.485,174.891,19.753,153.187
C03205=1086.367,76.884,437.502,174.889,19.752,153.187
C03206=1086.361,76.635,437.519,174.887,19.750,153.187
C03207=1086.356,76.386,437.536,174.885,19.748,153.187
C03208=1086.350,76.136,437.554,174.883,19.746,153.187
C03209=1086.344,75.887,437.571,174.882,19.744,153.187
C03210=1086.338,75.638,437.588,174.879,19.742,153.187
C03211=1086.333,75.388,437.605,174.878,19.741,153.187
C03212=1086.328,75.139,437.622,174.876,19.739,153.187
C03213=1086.321,74.890,437.639,174.874,19.737,153.187
C03214=1086.315,74.640,437.656,174.872,19.735,153.187
C03215=1086.310,74.391,437.674,174.871,19.733,153.187
C03216=1086.304,74.141,437.690,174.868,19.731,153.187
C03217=1086.298,73.892,437.708,174.867,19.729,153.187
C03218=1086.293,73.643,437.724,174.865,19.727,153.187
C03219=1086.287,73.394,437.741,174.863,19.726,153.187
C03220=1086.282,73.144,437.758,174.861,19.724,153.187
C03221=1086.277,72.895,437.775,174.860,19.722,153.186
C03222=1086.270,72.645,437.792,174.857,19.720,153.186
C03223=1086.265,72.396,437.809,174.856,19.718,153.186
C03224=1086.259,72.146,437.827,174.854,19.716,153.186
C03225=1086.253,71.897,437.843,174.852,19.714,153.186
C03226=1086.248,71.648,437.861,174.850,19.712,153.186
C03227=1086.242,71.399,437.877,174.849,19.711,153.186
C03228=1086.236,71.149,437.894,174.846,19.709,153.186
C03229=1086.231,70.900,437.911,174.845,19.707,153.186
C03230=1086.225,70.651,437.928,174.843,19.705,153.186
C03231=1086.220,70.401,437.944,174.841,19.703,153.186
C03232=1086.213,70.152,437.961,174.839,19.701,153.186
C03233=1086.208,69.902,437.979,174.838,19.699,153.186
C03234=1086.202,69.653,437.995,174.836,19.698,153.186
C03235=1086.196,69.404,438.012,174.834,19.695,153.186
C03236=1086.191,69.154,438.029,174.833,19.694,153.185
C03237=1086.185,68.905,438.046,174.830,19.692,153.185
C03238=1086.179,68.656,438.063,174.829,19.690,153.185
C03239=1086.174,68.406,438.079,174.827,19.688,153.185
C03240=1086.168,68.156,438.096,174.825,19.686,153.185
C03241=1086.162,67.907,438.112,174.823,19.684,153.185
C03242=1086.157,67.658,438.130,174.822,19.682,153.185
C03243=1086.151,67.409,438.146,174.819,19.680,153.185
C03244=1086.145,67.159,438.163,174.818,19.679,153.185
C03245=1086.139,66.910,438.180,174.816,19.677,153.185
C03246=1086.133,66.661,438.196,174.814,19.675,153.185
C03247=1086.128,66.411,438.213,174.812,19.673,153.185
C03248=1086.122,66.162,438.230,174.811,19.671,153.185
C03249=1086.117,65.912,438.246,174.809,19.669,153.185
C03250=1086.111,65.664,438.263,174.807,19.667,153.185
C03251=1086.106,65.414,438.280,174.806,19.666,153.185
C03252=1086.100,65.165,438.296,174.804,19.663,153.184
C03253=1086.094,64.915,438.313,174.802,19.662,153.184
C03254=1086.088,64.666,438.330,174.800,19.660,153.184
C03255=1086.082,64.416,438.346,174.799,19.658,153.184
C03256=1086.076,64.167,438.364,174.796,19.656,153.184
C03257=1086.070,63.917,438.380,174.795,19.654,153.184
C03258=1086.065,63.639,438.398,174.793,19.652,153.184
C03259=1086.058,63.361,438.417,174.790,19.650,153.184
C03260=1086.051,63.083,438.435,174.789,19.648,153.184
C03261=1086.045,62.805,438.453,174.787,19.646,153.184
C03262=1086.039,62.555,438.469,174.785,19.644,153.184
C03263=1086.033,62.306,438.486,174.783,19.642,153.184
C03264=1086.027,62.057,438.503,174.782,19.640,153.184
C03265=1086.022,61.807,438.519,174.779,19.638,153.184
C03266=1086.016,61.558,438.536,174.778,19.637,153.183
C03267=1086.010,61.309,438.552,174.776,19.634,153.183
C03268=1086.004,61.059,438.568,174.774,19.633,153.183
C03269=1085.998,60.810,438.584,174.772,19.631,153.183
C03270=1085.993,60.560,438.601,174.771,19.629,153.183
C03271=1085.987,60.311,438.618,174.769,19.627,153.183
C03272=1085.981,60.062,438.634,174.767,19.625,153.183
C03273=1085.975,59.812,438.650,174.766,19.623,153.183
C03274=1085.969,59.563,438.666,174.764,19.621,153.183
C03275=1085.964,59.313,438.683,174.762,19.620,153.183
C03276=1085.958,59.064,438.699,174.760,19.617,153.183
C03277=1085.952,58.815,438.716,174.759,19.616,153.183
C03278=1085.946,58.565,438.732,174.757,19.614,153.182
C03279=1085.940,58.316,438.748,174.755,19.612,153.182
C03280=1085.935,58.066,438.765,174.754,19.610,153.182
C03281=1085.929,57.817,438.781,174.751,19.608,153.182
C03282=1085.923,57.568,438.798,174.750,19.606,153.182
C03283=1085.917,57.318,438.814,174.748,19.604,153.182
C03284=1085.911,57.068,438.829,174.746,19.602,153.182
C03285=1085.905,56.819,438.846,174.745,19.601,153.182
C03286=1085.900,56.569,438.863,174.743,19.598,153.182
C03287=1085.894,56.320,438.879,174.741,19.597,153.182
C03288=1085.889,56.071,438.895,174.739,19.595,153.182
C03289=1085.883,55.822,438.911,174.738,19.593,153.182
C03290=1085.877,55.573,438.927,174.736,19.591,153.182
C03291=1085.871,55.323,438.943,174.734,19.589,153.181
C03292=1085.865,55.073,438.959,174.733,19.587,153.181
C03293=1085.860,54.824,438.976,174.731,19.585,153.181
C03294=1085.854,54.574,438.992,174.729,19.583,153.181
C03295=1085.848,54.325,439.008,174.727,19.581,153.181
C03296=1085.842,54.076,439.025,174.726,19.579,153.181
C03297=1085.837,53.827,439.040,174.723,19.577,153.181
C03298=1085.831,53.577,439.056,174.722,19.575,153.181
C03299=1085.825,53.328,439.072,174.721,19.573,153.181
C03300=1085.819,53.078,439.089,174.719,19.571,153.181
C03301=1085.814,52.829,439.105,174.717,19.569,153.181
C03302=1085.808,52.579,439.121,174.715,19.567,153.180
C03303=1085.803,52.330,439.137,174.714,19.565,153.180
C03304=1085.797,52.081,439.153,174.712,19.564,153.180
C03305=1085.791,51.831,439.169,174.710,19.561,153.180
C03306=1085.785,51.581,439.185,174.709,19.560,153.180
C03307=1085.779,51.332,439.201,174.707,19.557,153.180
C03308=1085.774,51.083,439.217,174.705,19.556,153.180
C03309=1085.768,50.834,439.233,174.703,19.553,153.180
C03310=1085.763,50.584,439.249,174.702,19.552,153.180
C03311=1085.757,50.335,439.265,174.700,19.550,153.180
C03312=1085.751,50.085,439.281,174.698,19.548,153.180
C03313=1085.746,49.835,439.297,174.697,19.546,153.179
C03314=1085.740,49.586,439.313,174.694,19.544,153.179
C03315=1085.734,49.337,439.330,174.693,19.542,153.179
C03316=1085.729,49.087,439.345,174.692,19.540,153.179
C03317=1085.723,48.838,439.361,174.690,19.538,153.179
C03318=1085.717,48.589,439.377,174.689,19.536,153.179
C03319=1085.712,48.339,439.393,174.686,19.534,153.179
C03320=1085.706,48.090,439.409,174.685,19.532,153.179
C03321=1085.700,47.840,439.425,174.684,19.530,153.179
C03322=1085.694,47.562,439.442,174.681,19.528,153.178
C03323=1085.688,47.283,439.461,174.679,19.525,153.178
C03324=1085.681,47.005,439.478,174.677,19.523,153.178
C03325=1085.675,46.727,439.495,174.676,19.521,153.178
C03326=1085.669,46.478,439.512,174.674,19.519,153.178
C03327=1085.664,46.228,439.527,174.672,19.517,153.178
C03328=1085.658,45.978,439.543,174.671,19.515,153.178
C03329=1085.653,45.729,439.559,174.669,19.513,153.178
C03330=1085.647,45.480,439.575,174.668,19.511,153.178
C03331=1085.641,45.230,439.590,174.665,19.509,153.177
C03332=1085.636,44.981,439.606,174.664,19.507,153.177
C03333=1085.630,44.731,439.622,174.663,19.505,153.177
C03334=1085.624,44.482,439.638,174.660,19.503,153.177
C03335=1085.619,44.232,439.653,174.659,19.501,153.177
C03336=1085.613,43.983,439.670,174.657,19.499,153.177
C03337=1085.607,43.733,439.685,174.656,19.497,153.177
C03338=1085.602,43.484,439.701,174.654,19.495,153.177
C03339=1085.596,43.234,439.717,174.652,19.493,153.177
C03340=1085.591,42.985,439.733,174.651,19.491,153.176
C03341=1085.584,42.735,439.748,174.649,19.490,153.176
C03342=1085.579,42.487,439.764,174.647,19.487,153.176
C03343=1085.573,42.237,439.779,174.646,19.485,153.176
C03344=1085.568,41.987,439.795,174.644,19.483,153.176
C03345=1085.562,41.738,439.811,174.642,19.481,153.176
C03346=1085.556,41.489,439.826,174.641,19.479,153.176
C03347=1085.550,41.239,439.842,174.639,19.477,153.176
C03348=1085.544,40.989,439.857,174.638,19.475,153.176
C03349=1085.539,40.740,439.872,174.636,19.473,153.176
C03350=1085.533,40.491,439.889,174.634,19.471,153.176
C03351=1085.527,40.241,439.904,174.633,19.469,153.175
C03352=1085.521,39.992,439.920,174.631,19.467,153.175
C03353=1085.516,39.742,439.935,174.629,19.465,153.175
C03354=1085.510,39.492,439.951,174.628,19.464,153.175
C03355=1085.505,39.244,439.967,174.626,19.461,153.175
C03356=1085.498,38.994,439.982,174.625,19.459,153.175
C03357=1085.493,38.744,439.997,174.622,19.457,153.175
C03358=1085.488,38.495,440.012,174.621,19.455,153.175
C03359=1085.482,38.246,440.028,174.620,19.454,153.175
C03360=1085.476,37.997,440.043,174.618,19.451,153.174
C03361=1085.470,37.747,440.059,174.616,19.449,153.174
C03362=1085.464,37.497,440.075,174.615,19.448,153.174
C03363=1085.458,37.248,440.090,174.613,19.445,153.174
C03364=1085.453,36.998,440.105,174.611,19.444,153.174
C03365=1085.447,36.748,440.121,174.609,19.441,153.174
C03366=1085.441,36.499,440.136,174.608,19.440,153.174
C03367=1085.436,36.250,440.151,174.607,19.438,153.174
C03368=1085.429,36.000,440.166,174.604,19.436,153.174
C03369=1085.424,35.751,440.181,174.603,19.434,153.173
C03370=1085.418,35.502,440.198,174.602,19.432,153.173
C03371=1085.412,35.252,440.213,174.600,19.430,153.173
C03372=1085.407,35.003,440.228,174.598,19.428,153.173
C03373=1085.400,34.753,440.243,174.597,19.426,153.173
C03374=1085.395,34.503,440.258,174.595,19.424,153.173
C03375=1085.389,34.255,440.274,174.593,19.422,153.173
C03376=1085.383,34.005,440.289,174.591,19.419,153.173
C03377=1085.378,33.756,440.304,174.590,19.418,153.173
C03378=1085.372,33.506,440.319,174.589,19.416,153.172
C03379=1085.366,33.256,440.335,174.586,19.414,153.172
C03380=1085.360,33.007,440.349,174.585,19.412,153.172
C03381=1085.355,32.757,440.365,174.584,19.410,153.172
C03382=1085.349,32.508,440.381,174.581,19.408,153.172
C03383=1085.343,32.259,440.396,174.580,19.406,153.172
C03384=1085.337,32.009,440.411,174.579,19.404,153.172
C03385=1085.331,31.760,440.426,174.577,19.402,153.172
C03386=1085.325,31.481,440.442,174.576,19.400,153.172
C03387=1085.319,31.203,440.460,174.573,19.397,153.171
C03388=1085.312,30.924,440.477,174.571,19.395,153.171
C03389=1085.306,30.646,440.493,174.570,19.393,153.171
C03390=1085.300,30.397,440.509,174.568,19.391,153.171
C03391=1085.294,30.147,440.524,174.566,19.389,153.171
C03392=1085.289,29.898,440.539,174.565,19.387,153.171
C03393=1085.283,29.649,440.554,174.563,19.385,153.171
C03394=1085.277,29.399,440.570,174.562,19.383,153.171
C03395=1085.271,29.150,440.584,174.560,19.381,153.170
C03396=1085.266,28.900,440.600,174.558,19.379,153.170
C03397=1085.260,28.651,440.615,174.557,19.377,153.170
C03398=1085.254,28.401,440.630,174.556,19.375,153.170
C03399=1085.248,28.152,440.645,174.553,19.373,153.170
C03400=1085.242,27.902,440.660,174.552,19.371,153.170
C03401=1085.237,27.653,440.675,174.551,19.369,153.170
C03402=1085.231,27.403,440.689,174.549,19.367,153.170
C03403=1085.226,27.153,440.704,174.547,19.365,153.170
C03404=1085.219,26.904,440.719,174.546,19.363,153.170
C03405=1085.214,26.655,440.734,174.544,19.361,153.169
C03406=1085.208,26.405,440.749,174.542,19.359,153.169
C03407=1085.202,26.156,440.764,174.541,19.357,153.169
C03408=1085.197,25.906,440.779,174.539,19.355,153.169
C03409=1085.190,25.656,440.794,174.538,19.353,153.169
C03410=1085.184,25.407,440.809,174.537,19.351,153.169
C03411=1085.179,25.157,440.824,174.534,19.349,153.169
C03412=1085.173,24.908,440.839,174.533,19.347,153.169
C03413=1085.167,24.659,440.854,174.532,19.345,153.168
C03414=1085.162,24.409,440.868,174.529,19.343,153.168
C03415=1085.156,24.159,440.883,174.528,19.341,153.168
C03416=1085.150,23.910,440.898,174.527,19.340,153.168
C03417=1085.144,23.660,440.913,174.525,19.337,153.168
C03418=1085.138,23.411,440.928,174.524,19.335,153.168
C03419=1085.133,23.162,440.943,174.522,19.334,153.168
C03420=1085.127,22.912,440.957,174.520,19.331,153.168
C03421=1085.121,22.663,440.972,174.519,19.329,153.168
C03422=1085.115,22.413,440.987,174.517,19.328,153.167
C03423=1085.109,22.164,441.002,174.515,19.325,153.167
C03424=1085.104,21.914,441.017,174.514,19.324,153.167
C03425=1085.098,21.665,441.031,174.513,19.322,153.167
C03426=1085.092,21.415,441.046,174.511,19.319,153.167
C03427=1085.087,21.166,441.061,174.509,19.317,153.167
C03428=1085.080,20.916,441.076,174.508,19.315,153.167
C03429=1085.075,20.666,441.090,174.507,19.313,153.167
C03430=1085.069,20.417,441.104,174.504,19.311,153.167
C03431=1085.063,20.167,441.120,174.503,19.309,153.166
C03432=1085.058,19.919,441.135,174.502,19.307,153.166
C03433=1085.052,19.668,441.149,174.500,19.305,153.166
C03434=1085.046,19.419,441.163,174.498,19.303,153.166
C03435=1085.040,19.169,441.179,174.497,19.302,153.166
C03436=1085.035,18.920,441.193,174.495,19.299,153.166
C03437=1085.029,18.671,441.207,174.494,19.297,153.166
C03438=1085.022,18.421,441.222,174.492,19.296,153.166
C03439=1085.017,18.172,441.236,174.490,19.293,153.165
C03440=1085.011,17.922,441.251,174.489,19.292,153.165
C03441=1085.006,17.673,441.266,174.487,19.290,153.165
C03442=1085.000,17.423,441.280,174.485,19.287,153.165
C03443=1084.994,17.173,441.295,174.484,19.286,153.165
C03444=1084.988,16.924,441.310,174.483,19.284,153.165
C03445=1084.982,16.674,441.324,174.482,19.282,153.165
C03446=1084.976,16.425,441.339,174.479,19.280,153.165
C03447=1084.971,16.175,441.353,174.478,19.277,153.165
C03448=1084.965,15.926,441.368,174.477,19.276,153.164
C03449=1084.959,15.677,441.383,174.475,19.273,153.164
C03450=1084.953,15.399,441.398,174.473,19.271,153.164
C03451=1084.946,15.123,441.414,174.471,19.269,153.164
C03452=1084.940,14.845,441.431,174.470,19.267,153.164
C03453=1084.933,14.568,441.446,174.468,19.265,153.164
C03454=1084.928,14.319,441.461,174.467,19.263,153.164
C03455=1084.922,14.070,441.476,174.465,19.261,153.163
C03456=1084.916,13.820,441.490,174.463,19.259,153.163
C03457=1084.910,13.571,441.504,174.462,19.257,153.163
C03458=1084.904,13.321,441.519,174.460,19.255,153.163
C03459=1084.898,13.072,441.533,174.458,19.253,153.163
C03460=1084.893,12.822,441.547,174.457,19.251,153.163
C03461=1084.886,12.572,441.562,174.456,19.249,153.163
C03462=1084.881,12.323,441.576,174.454,19.247,153.163
C03463=1084.875,12.074,441.590,174.452,19.245,153.163
C03464=1084.869,11.824,441.605,174.451,19.243,153.163
C03465=1084.863,11.575,441.619,174.449,19.242,153.162
C03466=1084.857,11.324,441.634,174.447,19.239,153.162
C03467=1084.851,11.076,441.648,174.446,19.237,153.162
C03468=1084.845,10.826,441.661,174.445,19.235,153.162
C03469=1084.839,10.576,441.676,174.443,19.233,153.162
C03470=1084.833,10.327,441.690,174.441,19.231,153.162
C03471=1084.828,10.077,441.704,174.440,19.229,153.162
C03472=1084.821,9.828,441.719,174.439,19.227,153.162
C03473=1084.816,9.578,441.733,174.436,19.225,153.162
C03474=1084.810,9.329,441.747,174.435,19.223,153.161
C03475=1084.804,9.079,441.762,174.434,19.222,153.161
C03476=1084.798,8.829,441.776,174.432,19.219,153.161
C03477=1084.793,8.580,441.790,174.431,19.217,153.161
C03478=1084.787,8.330,441.804,174.429,19.216,153.161
C03479=1084.780,8.081,441.818,174.428,19.214,153.161
C03480=1084.775,7.832,441.832,174.426,19.212,153.161
C03481=1084.769,7.582,441.846,174.424,19.210,153.161
C03482=1084.763,7.332,441.860,174.423,19.208,153.160
C03483=1084.757,7.083,441.875,174.422,19.206,153.160
C03484=1084.752,6.833,441.889,174.420,19.204,153.160
C03485=1084.746,6.583,441.903,174.418,19.202,153.160
C03486=1084.740,6.334,441.918,174.417,19.200,153.160
C03487=1084.734,6.085,441.931,174.415,19.197,153.160
C03488=1084.728,5.835,441.945,174.413,19.196,153.160
C03489=1084.722,5.586,441.960,174.412,19.194,153.160
C03490=1084.716,5.336,441.973,174.411,19.192,153.160
C03491=1084.711,5.087,441.987,174.409,19.190,153.160
C03492=1084.705,4.837,442.001,174.408,19.188,153.159
C03493=1084.699,4.587,442.016,174.406,19.186,153.159
C03494=1084.694,4.338,442.030,174.404,19.184,153.159
C03495=1084.687,4.089,442.043,174.403,19.182,153.159
C03496=1084.682,3.839,442.057,174.401,19.180,153.159
C03497=1084.676,3.589,442.072,174.400,19.178,153.159
C03498=1084.670,3.340,442.086,174.398,19.176,153.159
C03499=1084.665,3.090,442.100,174.397,19.174,153.159
C03500=1084.659,2.841,442.114,174.395,19.172,153.158
C03501=1084.653,2.591,442.127,174.394,19.170,153.158
C03502=1084.647,2.342,442.142,174.392,19.168,153.158
C03503=1084.641,2.092,442.156,174.391,19.166,153.158
C03504=1084.636,1.843,442.170,174.389,19.164,153.158
C03505=1084.630,1.593,442.184,174.388,19.162,153.158
C03506=1084.625,1.343,442.197,174.386,19.160,153.158
C03507=1084.618,1.093,442.211,174.385,19.158,153.158
C03508=1084.612,0.844,442.225,174.383,19.156,153.157
C03509=1084.607,0.595,442.239,174.381,19.154,153.157
C03510=1084.601,0.345,442.253,174.380,19.152,153.157
C03511=1084.596,0.096,442.267,174.379,19.150,153.157
C03512=1084.589,-0.154,442.280,174.378,19.148,153.157
C03513=1084.584,-0.403,442.294,174.375,19.146,153.157
C03514=1084.577,-0.679,442.310,174.374,19.144,153.157
C03515=1084.571,-0.954,442.326,174.372,19.142,153.157
C03516=1084.565,-1.229,442.341,174.371,19.140,153.156
C03517=1084.558,-1.504,442.355,174.369,19.137,153.156
C03518=1084.553,-1.753,442.369,174.367,19.135,153.156
C03519=1084.547,-2.003,442.383,174.366,19.133,153.156
C03520=1084.541,-2.252,442.396,174.365,19.131,153.156
C03521=1084.536,-2.502,442.410,174.363,19.129,153.156
C03522=1084.530,-2.751,442.425,174.361,19.127,153.156
C03523=1084.524,-3.000,442.439,174.360,19.125,153.156
C03524=1084.518,-3.250,442.452,174.359,19.124,153.155
C03525=1084.512,-3.500,442.466,174.357,19.121,153.155
C03526=1084.506,-3.749,442.480,174.355,19.120,153.155
C03527=1084.501,-3.999,442.493,174.354,19.118,153.155
C03528=1084.495,-4.248,442.507,174.353,19.116,153.155
C03529=1084.489,-4.497,442.521,174.350,19.114,153.155
C03530=1084.483,-4.748,442.535,174.349,19.112,153.155
C03531=1084.477,-4.998,442.547,174.348,19.110,153.155
C03532=1084.471,-5.247,442.561,174.347,19.108,153.155
C03533=1084.465,-5.496,442.574,174.345,19.107,153.155
C03534=1084.460,-5.746,442.588,174.343,19.104,153.154
C03535=1084.453,-5.995,442.602,174.342,19.102,153.154
C03536=1084.448,-6.245,442.615,174.340,19.100,153.154
C03537=1084.441,-6.495,442.629,174.339,19.098,153.154
C03538=1084.436,-6.744,442.643,174.337,19.096,153.154
C03539=1084.429,-6.994,442.656,174.336,19.094,153.154
C03540=1084.424,-7.243,442.670,174.334,19.093,153.154
C03541=1084.418,-7.492,442.683,174.333,19.091,153.154
C03542=1084.412,-7.742,442.697,174.331,19.089,153.154
C03543=1084.407,-7.992,442.711,174.330,19.087,153.153
C03544=1084.401,-8.241,442.724,174.328,19.085,153.153
C03545=1084.395,-8.491,442.737,174.327,19.083,153.153
C03546=1084.389,-8.741,442.751,174.325,19.081,153.153
C03547=1084.383,-8.991,442.765,174.323,19.079,153.153
C03548=1084.377,-9.240,442.778,174.322,19.077,153.153
C03549=1084.371,-9.489,442.792,174.321,19.076,153.153
C03550=1084.366,-9.739,442.805,174.320,19.073,153.153
C03551=1084.359,-9.989,442.818,174.318,19.071,153.152
C03552=1084.354,-10.238,442.832,174.316,19.069,153.152
C03553=1084.348,-10.487,442.845,174.315,19.067,153.152
C03554=1084.342,-10.737,442.859,174.313,19.066,153.152
C03555=1084.336,-10.987,442.871,174.311,19.063,153.152
C03556=1084.331,-11.236,442.885,174.310,19.062,153.152
C03557=1084.325,-11.486,442.899,174.309,19.060,153.152
C03558=1084.319,-11.735,442.912,174.308,19.058,153.152
C03559=1084.313,-11.985,442.926,174.305,19.056,153.152
C03560=1084.308,-12.235,442.939,174.304,19.054,153.151
C03561=1084.302,-12.484,442.952,174.303,19.052,153.151
C03562=1084.296,-12.734,442.966,174.301,19.050,153.151
C03563=1084.290,-12.983,442.979,174.300,19.048,153.151
C03564=1084.284,-13.233,442.992,174.298,19.046,153.151
C03565=1084.278,-13.482,443.006,174.297,19.044,153.151
C03566=1084.272,-13.732,443.019,174.295,19.042,153.151
C03567=1084.267,-13.982,443.032,174.294,19.040,153.151
C03568=1084.261,-14.231,443.045,174.292,19.038,153.151
C03569=1084.255,-14.481,443.059,174.291,19.036,153.151
C03570=1084.249,-14.730,443.072,174.289,19.034,153.150
C03571=1084.243,-14.980,443.085,174.288,19.033,153.150
C03572=1084.238,-15.229,443.099,174.287,19.031,153.150
C03573=1084.232,-15.479,443.112,174.284,19.029,153.150
C03574=1084.226,-15.728,443.125,174.283,19.027,153.150
C03575=1084.220,-15.978,443.139,174.282,19.025,153.150
C03576=1084.214,-16.228,443.151,174.281,19.023,153.150
C03577=1084.208,-16.477,443.164,174.279,19.022,153.150
C03578=1084.201,-16.751,443.179,174.277,19.019,153.150
C03579=1084.195,-17.025,443.193,174.276,19.017,153.150
C03580=1084.188,-17.298,443.208,174.274,19.015,153.149
C03581=1084.182,-17.571,443.222,174.272,19.013,153.149
C03582=1084.176,-17.820,443.236,174.271,19.011,153.149
C03583=1084.170,-18.070,443.248,174.269,19.009,153.149
C03584=1084.164,-18.319,443.262,174.268,19.007,153.149
C03585=1084.158,-18.569,443.274,174.266,19.005,153.149
C03586=1084.152,-18.819,443.287,174.265,19.004,153.149
C03587=1084.147,-19.069,443.301,174.264,19.002,153.149
C03588=1084.141,-19.318,443.314,174.261,19.000,153.149
C03589=1084.135,-19.567,443.327,174.260,18.998,153.148
C03590=1084.129,-19.817,443.340,174.259,18.996,153.148
C03591=1084.123,-20.067,443.353,174.258,18.994,153.148
C03592=1084.117,-20.317,443.366,174.256,18.993,153.148
C03593=1084.111,-20.566,443.379,174.254,18.990,153.148
C03594=1084.105,-20.816,443.392,174.253,18.988,153.148
C03595=1084.099,-21.065,443.405,174.251,18.986,153.148
C03596=1084.094,-21.315,443.418,174.250,18.985,153.148
C03597=1084.087,-21.564,443.432,174.249,18.983,153.148
C03598=1084.082,-21.814,443.444,174.246,18.981,153.148
C03599=1084.076,-22.063,443.457,174.245,18.979,153.147
C03600=1084.070,-22.313,443.470,174.244,18.977,153.147
C03601=1084.065,-22.563,443.483,174.243,18.975,153.147
C03602=1084.059,-22.812,443.496,174.241,18.974,153.147
C03603=1084.053,-23.062,443.509,174.239,18.971,153.147
C03604=1084.047,-23.311,443.522,174.238,18.970,153.147
C03605=1084.041,-23.561,443.534,174.237,18.968,153.147
C03606=1084.034,-23.811,443.548,174.235,18.966,153.147
C03607=1084.029,-24.061,443.561,174.234,18.964,153.147
C03608=1084.024,-24.310,443.573,174.232,18.962,153.147
C03609=1084.018,-24.559,443.586,174.230,18.960,153.146
C03610=1084.012,-24.809,443.599,174.229,18.958,153.146
C03611=1084.006,-25.059,443.611,174.228,18.956,153.146
C03612=1084.000,-25.308,443.625,174.226,18.955,153.146
C03613=1083.994,-25.558,443.637,174.225,18.953,153.146
C03614=1083.988,-25.808,443.651,174.223,18.951,153.146
C03615=1083.982,-26.058,443.664,174.222,18.949,153.146
C03616=1083.977,-26.307,443.676,174.220,18.947,153.146
C03617=1083.971,-26.556,443.689,174.219,18.945,153.146
C03618=1083.965,-26.806,443.702,174.218,18.944,153.146
C03619=1083.959,-27.056,443.714,174.216,18.942,153.145
C03620=1083.953,-27.305,443.727,174.214,18.939,153.145
C03621=1083.947,-27.555,443.740,174.213,18.938,153.145
C03622=1083.941,-27.805,443.753,174.211,18.936,153.145
C03623=1083.936,-28.054,443.765,174.210,18.934,153.145
C03624=1083.930,-28.303,443.778,174.209,18.932,153.145
C03625=1083.924,-28.553,443.791,174.207,18.930,153.145
C03626=1083.918,-28.803,443.803,174.205,18.929,153.145
C03627=1083.912,-29.052,443.816,174.204,18.927,153.145
C03628=1083.906,-29.302,443.829,174.202,18.925,153.145
C03629=1083.900,-29.552,443.841,174.201,18.923,153.145
C03630=1083.894,-29.802,443.854,174.200,18.922,153.145
C03631=1083.888,-30.050,443.867,174.198,18.920,153.145
C03632=1083.882,-30.300,443.879,174.196,18.918,153.144
C03633=1083.876,-30.550,443.892,174.195,18.916,153.144
C03634=1083.870,-30.800,443.904,174.194,18.914,153.144
C03635=1083.864,-31.050,443.917,174.192,18.912,153.144
C03636=1083.858,-31.299,443.930,174.191,18.911,153.144
C03637=1083.852,-31.548,443.942,174.189,18.908,153.144
C03638=1083.846,-31.798,443.955,174.187,18.907,153.144
C03639=1083.840,-32.048,443.967,174.186,18.905,153.144
C03640=1083.835,-32.298,443.980,174.185,18.903,153.144
C03641=1083.828,-32.547,443.993,174.183,18.902,153.144
